LIN {X 0,Y 504.867,Z 563.28,A -85,B 0,C 180,E1 5576.571,E2 5576.571} C_VEL
LIN {X 0,Y 504.82,Z 563.28,A -85,B 0,C 180,E1 5581.711,E2 5581.711} C_VEL
LIN {X 0,Y 504.782,Z 563.28,A -85,B 0,C 180,E1 5586.866,E2 5586.866} C_VEL
LIN {X 0,Y 504.734,Z 563.28,A -85,B 0,C 180,E1 5592.078,E2 5592.078} C_VEL
LIN {X 0,Y 504.643,Z 563.28,A -85,B 0,C 180,E1 5597.397,E2 5597.397} C_VEL
LIN {X 0,Y 504.494,Z 563.28,A -85,B 0,C 180,E1 5602.88,E2 5602.88} C_VEL
LIN {X 0,Y 504.391,Z 563.28,A -85,B 0,C 180,E1 5608.597,E2 5608.597} C_VEL
LIN {X 0,Y 504.485,Z 563.28,A -85,B 0,C 180,E1 5614.631,E2 5614.631} C_VEL
LIN {X 0,Y 504.229,Z 563.28,A -85,B 0,C 180,E1 5621.174,E2 5621.174} C_VEL
LIN {X 0,Y 504.156,Z 563.28,A -85,B 0,C 180,E1 5621.894,E2 5621.894} C_VEL
LIN {X 0,Y 500.156,Z 563.28,A -85,B 0,C 180,E1 5623.841,E2 5623.841} C_VEL
LIN {X 0,Y 496.221,Z 563.28,A -85,B 0,C 180,E1 5625.82,E2 5625.82} C_VEL
LIN {X 0,Y 496.453,Z 563.28,A -85,B 0,C 180,E1 5632.208,E2 5632.208} C_VEL
LIN {X 0,Y 496.52,Z 563.28,A -85,B 0,C 180,E1 5633.043,E2 5633.043} C_VEL
LIN {X 0,Y 514.224,Z 600.382,A -85,B 0,C 180,E1 5635.156,E2 5635.156} C_VEL
LIN {X 0,Y 512.783,Z 642.692,A -85,B 0,C 180,E1 5636.234,E2 5636.234} C_VEL
LIN {X 0,Y 510.259,Z 681.705,A -85,B 0,C 180,E1 5637.958,E2 5637.958} C_VEL
LIN {X 0,Y 507.477,Z 717.491,A -85,B 0,C 180,E1 5640.249,E2 5640.249} C_VEL
LIN {X 0,Y 504.31,Z 752.435,A -85,B 0,C 180,E1 5643.33,E2 5643.33} C_VEL
LIN {X 0,Y 501.653,Z 781.389,A -85,B 0,C 180,E1 5646.722,E2 5646.722} C_VEL
LIN {X 0,Y 499.587,Z 807.919,A -85,B 0,C 180,E1 5650.823,E2 5650.823} C_VEL
LIN {X 0,Y 498.227,Z 828.231,A -85,B 0,C 180,E1 5655.074,E2 5655.074} C_VEL
LIN {X 0,Y 497.609,Z 843.281,A -85,B 0,C 180,E1 5659.516,E2 5659.516} C_VEL
LIN {X 0,Y 497.334,Z 852.705,A -85,B 0,C 180,E1 5663.903,E2 5663.903} C_VEL
LIN {X 0,Y 497.217,Z 857.111,A -85,B 0,C 180,E1 5668.26,E2 5668.26} C_VEL
LIN {X 0,Y 497.291,Z 857.112,A -85,B 0,C 180,E1 5671.738,E2 5671.738} C_VEL
LIN {X 0,Y 497.33,Z 852.707,A -85,B 0,C 180,E1 5676.095,E2 5676.095} C_VEL
LIN {X 0,Y 497.429,Z 843.286,A -85,B 0,C 180,E1 5680.486,E2 5680.486} C_VEL
LIN {X 0,Y 498.149,Z 828.634,A -85,B 0,C 180,E1 5684.83,E2 5684.83} C_VEL
LIN {X 0,Y 499.508,Z 807.928,A -85,B 0,C 180,E1 5689.179,E2 5689.179} C_VEL
LIN {X 0,Y 501.629,Z 781.403,A -85,B 0,C 180,E1 5693.277,E2 5693.277} C_VEL
LIN {X 0,Y 504.374,Z 751.392,A -85,B 0,C 180,E1 5696.775,E2 5696.775} C_VEL
LIN {X 0,Y 507.446,Z 717.513,A -85,B 0,C 180,E1 5699.751,E2 5699.751} C_VEL
LIN {X 0,Y 510.334,Z 680.807,A -85,B 0,C 180,E1 5702.09,E2 5702.09} C_VEL
LIN {X 0,Y 512.765,Z 641.796,A -85,B 0,C 180,E1 5703.799,E2 5703.799} C_VEL
LIN {X 0,Y 513.861,Z 600.092,A -85,B 0,C 180,E1 5704.878,E2 5704.878} C_VEL
LIN {X 0,Y 496.473,Z 563.28,A -85,B 0,C 180,E1 5707.017,E2 5707.017} C_VEL
LIN {X 0,Y 496.268,Z 563.28,A -85,B 0,C 180,E1 5713.136,E2 5713.136} C_VEL
LIN {X 0,Y 496.316,Z 563.28,A -85,B 0,C 180,E1 5719.472,E2 5719.472} C_VEL
LIN {X 0,Y 496.36,Z 563.28,A -85,B 0,C 180,E1 5725.168,E2 5725.168} C_VEL
LIN {X 0,Y 496.405,Z 563.28,A -85,B 0,C 180,E1 5731.83,E2 5731.83} C_VEL
LIN {X 0,Y 496.526,Z 563.28,A -85,B 0,C 180,E1 5736.731,E2 5736.731} C_VEL
LIN {X 0,Y 496.737,Z 563.28,A -85,B 0,C 180,E1 5742.317,E2 5742.317} C_VEL
LIN {X 0,Y 496.762,Z 563.28,A -85,B 0,C 180,E1 5749.501,E2 5749.501} C_VEL
LIN {X 0,Y 496.987,Z 563.28,A -85,B 0,C 180,E1 5754.776,E2 5754.776} C_VEL
LIN {X 0,Y 497.058,Z 563.28,A -85,B 0,C 180,E1 5760.002,E2 5760.002} C_VEL
LIN {X 0,Y 496.985,Z 563.28,A -85,B 0,C 180,E1 5765.228,E2 5765.228} C_VEL
LIN {X 0,Y 496.817,Z 563.28,A -85,B 0,C 180,E1 5770.502,E2 5770.502} C_VEL
LIN {X 0,Y 496.757,Z 563.28,A -85,B 0,C 180,E1 5775.868,E2 5775.868} C_VEL
LIN {X 0,Y 496.651,Z 563.28,A -85,B 0,C 180,E1 5781.385,E2 5781.385} C_VEL
LIN {X 0,Y 496.463,Z 563.28,A -85,B 0,C 180,E1 5787.126,E2 5787.126} C_VEL
LIN {X 0,Y 496.548,Z 563.28,A -85,B 0,C 180,E1 5793.164,E2 5793.164} C_VEL
LIN {X 0,Y 496.39,Z 563.28,A -85,B 0,C 180,E1 5799.674,E2 5799.674} C_VEL
LIN {X 0,Y 496.273,Z 563.28,A -85,B 0,C 180,E1 5805.626,E2 5805.626} C_VEL
LIN {X 0,Y 496.467,Z 563.28,A -85,B 0,C 180,E1 5812.212,E2 5812.212} C_VEL
LIN {X 0,Y 496.517,Z 563.28,A -85,B 0,C 180,E1 5818.32,E2 5818.32} C_VEL
LIN {X 0,Y 496.487,Z 563.28,A -85,B 0,C 180,E1 5824.818,E2 5824.818} C_VEL
LIN {X 0,Y 496.629,Z 563.28,A -85,B 0,C 180,E1 5830.475,E2 5830.475} C_VEL
LIN {X 0,Y 496.875,Z 563.28,A -85,B 0,C 180,E1 5836.375,E2 5836.375} C_VEL
LIN {X 0,Y 496.906,Z 563.28,A -85,B 0,C 180,E1 5841.267,E2 5841.267} C_VEL
LIN {X 0,Y 497.111,Z 563.28,A -85,B 0,C 180,E1 5846.52,E2 5846.52} C_VEL
LIN {X 0,Y 497.235,Z 563.28,A -85,B 0,C 180,E1 5851.74,E2 5851.74} C_VEL
LIN {X 0,Y 496.994,Z 563.28,A -85,B 0,C 180,E1 5856.977,E2 5856.977} C_VEL
LIN {X 0,Y 496.771,Z 563.28,A -85,B 0,C 180,E1 5863.576,E2 5863.576} C_VEL
LIN {X 0,Y 496.648,Z 563.28,A -85,B 0,C 180,E1 5869.624,E2 5869.624} C_VEL
LIN {X 0,Y 496.506,Z 563.28,A -85,B 0,C 180,E1 5875.183,E2 5875.183} C_VEL
LIN {X 0,Y 496.317,Z 563.28,A -85,B 0,C 180,E1 5881.643,E2 5881.643} C_VEL
LIN {X 0,Y 496.45,Z 563.28,A -85,B 0,C 180,E1 5887.785,E2 5887.785} C_VEL
LIN {X 0,Y 496.341,Z 563.28,A -85,B 0,C 180,E1 5894.369,E2 5894.369} C_VEL
LIN {X 0,Y 496.34,Z 563.28,A -85,B 0,C 180,E1 5900.322,E2 5900.322} C_VEL
LIN {X 0,Y 496.337,Z 563.28,A -85,B 0,C 180,E1 5906.82,E2 5906.82} C_VEL
LIN {X 0,Y 496.455,Z 563.28,A -85,B 0,C 180,E1 5912.873,E2 5912.873} C_VEL
LIN {X 0,Y 496.667,Z 563.28,A -85,B 0,C 180,E1 5918.616,E2 5918.616} C_VEL
LIN {X 0,Y 496.65,Z 563.28,A -85,B 0,C 180,E1 5924.128,E2 5924.128} C_VEL
LIN {X 0,Y 496.761,Z 563.28,A -85,B 0,C 180,E1 5929.497,E2 5929.497} C_VEL
LIN {X 0,Y 497.004,Z 563.28,A -85,B 0,C 180,E1 5934.772,E2 5934.772} C_VEL
LIN {X 0,Y 497.072,Z 563.28,A -85,B 0,C 180,E1 5939.998,E2 5939.998} C_VEL
LIN {X 0,Y 496.994,Z 563.28,A -85,B 0,C 180,E1 5945.224,E2 5945.224} C_VEL
LIN {X 0,Y 496.867,Z 563.28,A -85,B 0,C 180,E1 5950.497,E2 5950.497} C_VEL
LIN {X 0,Y 496.741,Z 563.28,A -85,B 0,C 180,E1 5955.865,E2 5955.865} C_VEL
LIN {X 0,Y 496.644,Z 563.28,A -85,B 0,C 180,E1 5961.381,E2 5961.381} C_VEL
LIN {X 0,Y 496.455,Z 563.28,A -85,B 0,C 180,E1 5967.123,E2 5967.123} C_VEL
LIN {X 0,Y 496.554,Z 563.28,A -85,B 0,C 180,E1 5973.16,E2 5973.16} C_VEL
LIN {X 0,Y 496.352,Z 563.28,A -85,B 0,C 180,E1 5979.673,E2 5979.673} C_VEL
LIN {X 0,Y 496.221,Z 563.28,A -85,B 0,C 180,E1 5985.82,E2 5985.82} C_VEL
LIN {X 0,Y 492.298,Z 563.28,A -85,B 0,C 180,E1 5987.795,E2 5987.795} C_VEL
LIN {X 0,Y 488.41,Z 563.28,A -85,B 0,C 180,E1 5989.801,E2 5989.801} C_VEL
LIN {X 0,Y 488.571,Z 563.784,A -85,B 0,C 180,E1 5992.379,E2 5992.379} C_VEL
LIN {X 0,Y 507.767,Z 604.447,A -85,B 0,C 180,E1 5994.736,E2 5994.736} C_VEL
LIN {X 0,Y 506.121,Z 643.782,A -85,B 0,C 180,E1 5995.777,E2 5995.777} C_VEL
LIN {X 0,Y 503.313,Z 683.897,A -85,B 0,C 180,E1 5997.593,E2 5997.593} C_VEL
LIN {X 0,Y 500.324,Z 718.929,A -85,B 0,C 180,E1 5999.905,E2 5999.905} C_VEL
LIN {X 0,Y 496.964,Z 753.499,A -85,B 0,C 180,E1 6003.018,E2 6003.018} C_VEL
LIN {X 0,Y 494.007,Z 783.215,A -85,B 0,C 180,E1 6006.602,E2 6006.602} C_VEL
LIN {X 0,Y 491.844,Z 807.92,A -85,B 0,C 180,E1 6010.509,E2 6010.509} C_VEL
LIN {X 0,Y 490.4,Z 828.252,A -85,B 0,C 180,E1 6014.837,E2 6014.837} C_VEL
LIN {X 0,Y 489.736,Z 843.28,A -85,B 0,C 180,E1 6019.345,E2 6019.345} C_VEL
LIN {X 0,Y 489.443,Z 852.701,A -85,B 0,C 180,E1 6023.804,E2 6023.804} C_VEL
LIN {X 0,Y 489.315,Z 857.112,A -85,B 0,C 180,E1 6028.232,E2 6028.232} C_VEL
LIN {X 0,Y 489.385,Z 857.113,A -85,B 0,C 180,E1 6031.766,E2 6031.766} C_VEL
LIN {X 0,Y 489.435,Z 852.703,A -85,B 0,C 180,E1 6036.194,E2 6036.194} C_VEL
LIN {X 0,Y 489.564,Z 843.284,A -85,B 0,C 180,E1 6040.657,E2 6040.657} C_VEL
LIN {X 0,Y 490.259,Z 830.078,A -85,B 0,C 180,E1 6044.71,E2 6044.71} C_VEL
LIN {X 0,Y 491.631,Z 810.331,A -85,B 0,C 180,E1 6049.033,E2 6049.033} C_VEL
LIN {X 0,Y 493.663,Z 786.566,A -85,B 0,C 180,E1 6052.937,E2 6052.937} C_VEL
LIN {X 0,Y 496.595,Z 756.593,A -85,B 0,C 180,E1 6056.655,E2 6056.655} C_VEL
LIN {X 0,Y 499.865,Z 723.287,A -85,B 0,C 180,E1 6059.749,E2 6059.749} C_VEL
LIN {X 0,Y 503.147,Z 687.121,A -85,B 0,C 180,E1 6062.227,E2 6062.227} C_VEL
LIN {X 0,Y 505.785,Z 649.282,A -85,B 0,C 180,E1 6064.01,E2 6064.01} C_VEL
LIN {X 0,Y 507.694,Z 611.444,A -85,B 0,C 180,E1 6065.125,E2 6065.125} C_VEL
LIN {X 0,Y 507.191,Z 602.422,A -85,B 0,C 180,E1 6065.351,E2 6065.351} C_VEL
LIN {X 0,Y 488.543,Z 563.28,A -85,B 0,C 180,E1 6067.702,E2 6067.702} C_VEL
LIN {X 0,Y 488.399,Z 563.28,A -85,B 0,C 180,E1 6074.717,E2 6074.717} C_VEL
LIN {X 0,Y 488.385,Z 563.28,A -85,B 0,C 180,E1 6080.573,E2 6080.573} C_VEL
LIN {X 0,Y 488.423,Z 563.28,A -85,B 0,C 180,E1 6086.529,E2 6086.529} C_VEL
LIN {X 0,Y 488.502,Z 563.28,A -85,B 0,C 180,E1 6092.399,E2 6092.399} C_VEL
LIN {X 0,Y 488.681,Z 563.28,A -85,B 0,C 180,E1 6098.253,E2 6098.253} C_VEL
LIN {X 0,Y 488.72,Z 563.28,A -85,B 0,C 180,E1 6103.868,E2 6103.868} C_VEL
LIN {X 0,Y 488.839,Z 563.28,A -85,B 0,C 180,E1 6109.328,E2 6109.328} C_VEL
LIN {X 0,Y 489.075,Z 563.28,A -85,B 0,C 180,E1 6114.691,E2 6114.691} C_VEL
LIN {X 0,Y 489.158,Z 563.28,A -85,B 0,C 180,E1 6120.002,E2 6120.002} C_VEL
LIN {X 0,Y 489.069,Z 563.28,A -85,B 0,C 180,E1 6125.313,E2 6125.313} C_VEL
LIN {X 0,Y 488.899,Z 563.28,A -85,B 0,C 180,E1 6130.674,E2 6130.674} C_VEL
LIN {X 0,Y 488.786,Z 563.28,A -85,B 0,C 180,E1 6136.856,E2 6136.856} C_VEL
LIN {X 0,Y 488.676,Z 563.28,A -85,B 0,C 180,E1 6142.124,E2 6142.124} C_VEL
LIN {X 0,Y 488.545,Z 563.28,A -85,B 0,C 180,E1 6147.603,E2 6147.603} C_VEL
LIN {X 0,Y 488.608,Z 563.28,A -85,B 0,C 180,E1 6153.775,E2 6153.775} C_VEL
LIN {X 0,Y 488.471,Z 563.28,A -85,B 0,C 180,E1 6159.439,E2 6159.439} C_VEL
LIN {X 0,Y 488.365,Z 563.28,A -85,B 0,C 180,E1 6165.292,E2 6165.292} C_VEL
LIN {X 0,Y 488.529,Z 563.28,A -85,B 0,C 180,E1 6171.847,E2 6171.847} C_VEL
LIN {X 0,Y 488.618,Z 563.28,A -85,B 0,C 180,E1 6178.332,E2 6178.332} C_VEL
LIN {X 0,Y 488.526,Z 563.28,A -85,B 0,C 180,E1 6184.378,E2 6184.378} C_VEL
LIN {X 0,Y 488.714,Z 563.28,A -85,B 0,C 180,E1 6190.145,E2 6190.145} C_VEL
LIN {X 0,Y 488.91,Z 563.28,A -85,B 0,C 180,E1 6195.706,E2 6195.706} C_VEL
LIN {X 0,Y 489.001,Z 563.28,A -85,B 0,C 180,E1 6201.125,E2 6201.125} C_VEL
LIN {X 0,Y 489.2,Z 563.28,A -85,B 0,C 180,E1 6206.464,E2 6206.464} C_VEL
LIN {X 0,Y 489.324,Z 563.28,A -85,B 0,C 180,E1 6211.768,E2 6211.768} C_VEL
LIN {X 0,Y 489.068,Z 563.28,A -85,B 0,C 180,E1 6217.09,E2 6217.09} C_VEL
LIN {X 0,Y 488.878,Z 563.28,A -85,B 0,C 180,E1 6222.479,E2 6222.479} C_VEL
LIN {X 0,Y 488.759,Z 563.28,A -85,B 0,C 180,E1 6227.984,E2 6227.984} C_VEL
LIN {X 0,Y 488.634,Z 563.28,A -85,B 0,C 180,E1 6233.671,E2 6233.671} C_VEL
LIN {X 0,Y 488.384,Z 563.28,A -85,B 0,C 180,E1 6240.099,E2 6240.099} C_VEL
LIN {X 0,Y 488.463,Z 563.28,A -85,B 0,C 180,E1 6245.943,E2 6245.943} C_VEL
LIN {X 0,Y 488.394,Z 563.28,A -85,B 0,C 180,E1 6252.136,E2 6252.136} C_VEL
LIN {X 0,Y 488.423,Z 563.28,A -85,B 0,C 180,E1 6257.86,E2 6257.86} C_VEL
LIN {X 0,Y 488.396,Z 563.28,A -85,B 0,C 180,E1 6264.051,E2 6264.051} C_VEL
LIN {X 0,Y 488.431,Z 563.28,A -85,B 0,C 180,E1 6270.373,E2 6270.373} C_VEL
LIN {X 0,Y 488.653,Z 563.28,A -85,B 0,C 180,E1 6276.329,E2 6276.329} C_VEL
LIN {X 0,Y 488.83,Z 563.28,A -85,B 0,C 180,E1 6282.018,E2 6282.018} C_VEL
LIN {X 0,Y 488.84,Z 563.28,A -85,B 0,C 180,E1 6289.325,E2 6289.325} C_VEL
LIN {X 0,Y 489.092,Z 563.28,A -85,B 0,C 180,E1 6294.687,E2 6294.687} C_VEL
LIN {X 0,Y 489.171,Z 563.28,A -85,B 0,C 180,E1 6299.998,E2 6299.998} C_VEL
LIN {X 0,Y 489.078,Z 563.28,A -85,B 0,C 180,E1 6305.309,E2 6305.309} C_VEL
LIN {X 0,Y 488.942,Z 563.28,A -85,B 0,C 180,E1 6310.669,E2 6310.669} C_VEL
LIN {X 0,Y 488.761,Z 563.28,A -85,B 0,C 180,E1 6316.841,E2 6316.841} C_VEL
LIN {X 0,Y 488.666,Z 563.28,A -85,B 0,C 180,E1 6322.116,E2 6322.116} C_VEL
LIN {X 0,Y 488.537,Z 563.28,A -85,B 0,C 180,E1 6327.599,E2 6327.599} C_VEL
LIN {X 0,Y 488.612,Z 563.28,A -85,B 0,C 180,E1 6333.77,E2 6333.77} C_VEL
LIN {X 0,Y 488.435,Z 563.28,A -85,B 0,C 180,E1 6339.432,E2 6339.432} C_VEL
LIN {X 0,Y 488.281,Z 563.28,A -85,B 0,C 180,E1 6345.814,E2 6345.814} C_VEL
LIN {X 0,Y 488.41,Z 563.28,A -85,B 0,C 180,E1 6349.801,E2 6349.801} C_VEL
LIN {X 0,Y 487.978,Z 566.18,A -85,B 0,C 180,E1 6350.996,E2 6350.996} C_VEL
LIN {X 0,Y 488.177,Z 576.133,A -85,B 0,C 180,E1 6352.344,E2 6352.344} C_VEL
LIN {X 0,Y 490.346,Z 583.192,A -85,B 0,C 180,E1 6352.886,E2 6352.886} C_VEL
LIN {X 0,Y 501.242,Z 607.303,A -85,B 0,C 180,E1 6354.273,E2 6354.273} C_VEL
LIN {X 0,Y 499.283,Z 646.915,A -85,B 0,C 180,E1 6355.391,E2 6355.391} C_VEL
LIN {X 0,Y 496.205,Z 687.92,A -85,B 0,C 180,E1 6357.329,E2 6357.329} C_VEL
LIN {X 0,Y 492.71,Z 724.764,A -85,B 0,C 180,E1 6359.904,E2 6359.904} C_VEL
LIN {X 0,Y 489.37,Z 756.878,A -85,B 0,C 180,E1 6362.954,E2 6362.954} C_VEL
LIN {X 0,Y 486.217,Z 786.547,A -85,B 0,C 180,E1 6366.689,E2 6366.689} C_VEL
LIN {X 0,Y 483.93,Z 811.51,A -85,B 0,C 180,E1 6370.887,E2 6370.887} C_VEL
LIN {X 0,Y 482.505,Z 830.074,A -85,B 0,C 180,E1 6375.047,E2 6375.047} C_VEL
LIN {X 0,Y 481.795,Z 844.724,A -85,B 0,C 180,E1 6379.743,E2 6379.743} C_VEL
LIN {X 0,Y 481.41,Z 854.003,A -85,B 0,C 180,E1 6384.603,E2 6384.603} C_VEL
LIN {X 0,Y 481.427,Z 857.113,A -85,B 0,C 180,E1 6388.203,E2 6388.203} C_VEL
LIN {X 0,Y 481.485,Z 857.114,A -85,B 0,C 180,E1 6391.795,E2 6391.795} C_VEL
LIN {X 0,Y 481.55,Z 852.699,A -85,B 0,C 180,E1 6396.296,E2 6396.296} C_VEL
LIN {X 0,Y 481.701,Z 843.283,A -85,B 0,C 180,E1 6400.833,E2 6400.833} C_VEL
LIN {X 0,Y 482.465,Z 830.081,A -85,B 0,C 180,E1 6404.953,E2 6404.953} C_VEL
LIN {X 0,Y 484.091,Z 809.135,A -85,B 0,C 180,E1 6409.578,E2 6409.578} C_VEL
LIN {X 0,Y 486.353,Z 784.891,A -85,B 0,C 180,E1 6413.544,E2 6413.544} C_VEL
LIN {X 0,Y 489.526,Z 755.489,A -85,B 0,C 180,E1 6417.203,E2 6417.203} C_VEL
LIN {X 0,Y 493.015,Z 722.001,A -85,B 0,C 180,E1 6420.317,E2 6420.317} C_VEL
LIN {X 0,Y 496.415,Z 685.825,A -85,B 0,C 180,E1 6422.783,E2 6422.783} C_VEL
LIN {X 0,Y 499.341,Z 645.989,A -85,B 0,C 180,E1 6424.646,E2 6424.646} C_VEL
LIN {X 0,Y 500.914,Z 605.537,A -85,B 0,C 180,E1 6425.791,E2 6425.791} C_VEL
LIN {X 0,Y 480.578,Z 563.28,A -85,B 0,C 180,E1 6428.392,E2 6428.392} C_VEL
LIN {X 0,Y 480.437,Z 563.28,A -85,B 0,C 180,E1 6433.75,E2 6433.75} C_VEL
LIN {X 0,Y 480.462,Z 563.28,A -85,B 0,C 180,E1 6438.917,E2 6438.917} C_VEL
LIN {X 0,Y 480.44,Z 563.28,A -85,B 0,C 180,E1 6444.748,E2 6444.748} C_VEL
LIN {X 0,Y 480.493,Z 563.28,A -85,B 0,C 180,E1 6449.838,E2 6449.838} C_VEL
LIN {X 0,Y 480.662,Z 563.28,A -85,B 0,C 180,E1 6455.915,E2 6455.915} C_VEL
LIN {X 0,Y 480.872,Z 563.28,A -85,B 0,C 180,E1 6461.714,E2 6461.714} C_VEL
LIN {X 0,Y 480.785,Z 563.28,A -85,B 0,C 180,E1 6467.31,E2 6467.31} C_VEL
LIN {X 0,Y 481.133,Z 563.28,A -85,B 0,C 180,E1 6472.795,E2 6472.795} C_VEL
LIN {X 0,Y 481.416,Z 563.28,A -85,B 0,C 180,E1 6478.206,E2 6478.206} C_VEL
LIN {X 0,Y 481.297,Z 563.28,A -85,B 0,C 180,E1 6483.597,E2 6483.597} C_VEL
LIN {X 0,Y 481.064,Z 563.28,A -85,B 0,C 180,E1 6489.025,E2 6489.025} C_VEL
LIN {X 0,Y 480.976,Z 563.28,A -85,B 0,C 180,E1 6494.538,E2 6494.538} C_VEL
LIN {X 0,Y 480.827,Z 563.28,A -85,B 0,C 180,E1 6500.197,E2 6500.197} C_VEL
LIN {X 0,Y 480.651,Z 563.28,A -85,B 0,C 180,E1 6506.076,E2 6506.076} C_VEL
LIN {X 0,Y 480.66,Z 563.28,A -85,B 0,C 180,E1 6512.258,E2 6512.258} C_VEL
LIN {X 0,Y 480.585,Z 563.28,A -85,B 0,C 180,E1 6518.904,E2 6518.904} C_VEL
LIN {X 0,Y 480.406,Z 563.28,A -85,B 0,C 180,E1 6523.744,E2 6523.744} C_VEL
LIN {X 0,Y 480.469,Z 563.28,A -85,B 0,C 180,E1 6528.92,E2 6528.92} C_VEL
LIN {X 0,Y 480.628,Z 563.28,A -85,B 0,C 180,E1 6534.719,E2 6534.719} C_VEL
LIN {X 0,Y 480.653,Z 563.28,A -85,B 0,C 180,E1 6539.847,E2 6539.847} C_VEL
LIN {X 0,Y 480.604,Z 563.28,A -85,B 0,C 180,E1 6545.911,E2 6545.911} C_VEL
LIN {X 0,Y 480.82,Z 563.28,A -85,B 0,C 180,E1 6551.71,E2 6551.71} C_VEL
LIN {X 0,Y 481.01,Z 563.28,A -85,B 0,C 180,E1 6557.315,E2 6557.315} C_VEL
LIN {X 0,Y 481.09,Z 563.28,A -85,B 0,C 180,E1 6562.793,E2 6562.793} C_VEL
LIN {X 0,Y 481.194,Z 563.28,A -85,B 0,C 180,E1 6568.204,E2 6568.204} C_VEL
LIN {X 0,Y 481.212,Z 563.28,A -85,B 0,C 180,E1 6573.597,E2 6573.597} C_VEL
LIN {X 0,Y 481.043,Z 563.28,A -85,B 0,C 180,E1 6579.025,E2 6579.025} C_VEL
LIN {X 0,Y 480.919,Z 563.28,A -85,B 0,C 180,E1 6584.539,E2 6584.539} C_VEL
LIN {X 0,Y 480.787,Z 563.28,A -85,B 0,C 180,E1 6590.198,E2 6590.198} C_VEL
LIN {X 0,Y 480.615,Z 563.28,A -85,B 0,C 180,E1 6596.077,E2 6596.077} C_VEL
LIN {X 0,Y 480.505,Z 563.28,A -85,B 0,C 180,E1 6602.269,E2 6602.269} C_VEL
LIN {X 0,Y 480.583,Z 563.28,A -85,B 0,C 180,E1 6608.903,E2 6608.903} C_VEL
LIN {X 0,Y 480.47,Z 563.28,A -85,B 0,C 180,E1 6613.749,E2 6613.749} C_VEL
LIN {X 0,Y 480.48,Z 563.28,A -85,B 0,C 180,E1 6618.918,E2 6618.918} C_VEL
LIN {X 0,Y 480.443,Z 563.28,A -85,B 0,C 180,E1 6624.75,E2 6624.75} C_VEL
LIN {X 0,Y 480.501,Z 563.28,A -85,B 0,C 180,E1 6629.834,E2 6629.834} C_VEL
LIN {X 0,Y 480.686,Z 563.28,A -85,B 0,C 180,E1 6635.912,E2 6635.912} C_VEL
LIN {X 0,Y 480.889,Z 563.28,A -85,B 0,C 180,E1 6641.71,E2 6641.71} C_VEL
LIN {X 0,Y 480.775,Z 563.28,A -85,B 0,C 180,E1 6647.306,E2 6647.306} C_VEL
LIN {X 0,Y 481.112,Z 563.28,A -85,B 0,C 180,E1 6653.004,E2 6653.004} C_VEL
LIN {X 0,Y 481.434,Z 563.28,A -85,B 0,C 180,E1 6658.202,E2 6658.202} C_VEL
LIN {X 0,Y 481.264,Z 563.28,A -85,B 0,C 180,E1 6663.593,E2 6663.593} C_VEL
LIN {X 0,Y 481.073,Z 563.28,A -85,B 0,C 180,E1 6669.021,E2 6669.021} C_VEL
LIN {X 0,Y 480.971,Z 563.28,A -85,B 0,C 180,E1 6674.534,E2 6674.534} C_VEL
LIN {X 0,Y 480.819,Z 563.28,A -85,B 0,C 180,E1 6680.193,E2 6680.193} C_VEL
LIN {X 0,Y 480.639,Z 563.28,A -85,B 0,C 180,E1 6686.072,E2 6686.072} C_VEL
LIN {X 0,Y 480.658,Z 563.28,A -85,B 0,C 180,E1 6692.254,E2 6692.254} C_VEL
LIN {X 0,Y 480.607,Z 563.28,A -85,B 0,C 180,E1 6698.283,E2 6698.283} C_VEL
LIN {X 0,Y 480.373,Z 563.28,A -85,B 0,C 180,E1 6703.737,E2 6703.737} C_VEL
LIN {X 0,Y 480.416,Z 563.28,A -85,B 0,C 180,E1 6709.804,E2 6709.804} C_VEL
LIN {X 0,Y 480.623,Z 564,A -85,B 0,C 180,E1 6711.655,E2 6711.655} C_VEL
LIN {X 0,Y 490.346,Z 583.192,A -85,B 0,C 180,E1 6712.886,E2 6712.886} C_VEL
LIN {X 0,Y 493.821,Z 595.133,A -85,B 0,C 180,E1 6713.4,E2 6713.4} C_VEL
LIN {X 0,Y 494.395,Z 616.987,A -85,B 0,C 180,E1 6713.952,E2 6713.952} C_VEL
LIN {X 0,Y 491.949,Z 657.63,A -85,B 0,C 180,E1 6715.296,E2 6715.296} C_VEL
LIN {X 0,Y 488.506,Z 697.035,A -85,B 0,C 180,E1 6717.407,E2 6717.407} C_VEL
LIN {X 0,Y 484.975,Z 731.703,A -85,B 0,C 180,E1 6720.03,E2 6720.03} C_VEL
LIN {X 0,Y 481.133,Z 765.214,A -85,B 0,C 180,E1 6723.468,E2 6723.468} C_VEL
LIN {X 0,Y 478.108,Z 792.986,A -85,B 0,C 180,E1 6727.3,E2 6727.3} C_VEL
LIN {X 0,Y 475.843,Z 816.208,A -85,B 0,C 180,E1 6731.51,E2 6731.51} C_VEL
LIN {X 0,Y 474.304,Z 835.931,A -85,B 0,C 180,E1 6736.472,E2 6736.472} C_VEL
LIN {X 0,Y 473.778,Z 847.752,A -85,B 0,C 180,E1 6740.865,E2 6740.865} C_VEL
LIN {X 0,Y 473.521,Z 854.003,A -85,B 0,C 180,E1 6744.513,E2 6744.513} C_VEL
LIN {X 0,Y 473.524,Z 857.113,A -85,B 0,C 180,E1 6748.173,E2 6748.173} C_VEL
LIN {X 0,Y 473.579,Z 857.114,A -85,B 0,C 180,E1 6751.825,E2 6751.825} C_VEL
LIN {X 0,Y 473.641,Z 852.696,A -85,B 0,C 180,E1 6756.401,E2 6756.401} C_VEL
LIN {X 0,Y 473.865,Z 843.282,A -85,B 0,C 180,E1 6761.014,E2 6761.014} C_VEL
LIN {X 0,Y 474.677,Z 830.084,A -85,B 0,C 180,E1 6765.204,E2 6765.204} C_VEL
LIN {X 0,Y 476.439,Z 809.132,A -85,B 0,C 180,E1 6769.905,E2 6769.905} C_VEL
LIN {X 0,Y 478.97,Z 784.467,A -85,B 0,C 180,E1 6773.991,E2 6773.991} C_VEL
LIN {X 0,Y 482.347,Z 755.059,A -85,B 0,C 180,E1 6777.694,E2 6777.694} C_VEL
LIN {X 0,Y 486.177,Z 720.586,A -85,B 0,C 180,E1 6780.895,E2 6780.895} C_VEL
LIN {X 0,Y 489.749,Z 684.504,A -85,B 0,C 180,E1 6783.352,E2 6783.352} C_VEL
LIN {X 0,Y 492.928,Z 643.347,A -85,B 0,C 180,E1 6785.27,E2 6785.27} C_VEL
LIN {X 0,Y 494.202,Z 607.589,A -85,B 0,C 180,E1 6786.305,E2 6786.305} C_VEL
LIN {X 0,Y 472.752,Z 564.557,A -85,B 0,C 180,E1 6789.087,E2 6789.087} C_VEL
LIN {X 0,Y 472.592,Z 563.28,A -85,B 0,C 180,E1 6789.255,E2 6789.255} C_VEL
LIN {X 0,Y 472.456,Z 563.28,A -85,B 0,C 180,E1 6795.362,E2 6795.362} C_VEL
LIN {X 0,Y 472.499,Z 563.28,A -85,B 0,C 180,E1 6800.306,E2 6800.306} C_VEL
LIN {X 0,Y 472.498,Z 563.28,A -85,B 0,C 180,E1 6806.134,E2 6806.134} C_VEL
LIN {X 0,Y 472.615,Z 563.28,A -85,B 0,C 180,E1 6811.387,E2 6811.387} C_VEL
LIN {X 0,Y 472.85,Z 563.28,A -85,B 0,C 180,E1 6817.738,E2 6817.738} C_VEL
LIN {X 0,Y 472.904,Z 563.28,A -85,B 0,C 180,E1 6823.313,E2 6823.313} C_VEL
LIN {X 0,Y 472.97,Z 563.28,A -85,B 0,C 180,E1 6828.966,E2 6828.966} C_VEL
LIN {X 0,Y 473.25,Z 563.28,A -85,B 0,C 180,E1 6834.513,E2 6834.513} C_VEL
LIN {X 0,Y 473.363,Z 563.28,A -85,B 0,C 180,E1 6840.002,E2 6840.002} C_VEL
LIN {X 0,Y 473.237,Z 563.28,A -85,B 0,C 180,E1 6845.491,E2 6845.491} C_VEL
LIN {X 0,Y 473.06,Z 563.28,A -85,B 0,C 180,E1 6851.036,E2 6851.036} C_VEL
LIN {X 0,Y 472.956,Z 563.28,A -85,B 0,C 180,E1 6856.831,E2 6856.831} C_VEL
LIN {X 0,Y 472.824,Z 563.28,A -85,B 0,C 180,E1 6862.52,E2 6862.52} C_VEL
LIN {X 0,Y 472.687,Z 563.28,A -85,B 0,C 180,E1 6868.613,E2 6868.613} C_VEL
LIN {X 0,Y 472.727,Z 563.28,A -85,B 0,C 180,E1 6875.072,E2 6875.072} C_VEL
LIN {X 0,Y 472.543,Z 563.28,A -85,B 0,C 180,E1 6879.969,E2 6879.969} C_VEL
LIN {X 0,Y 472.424,Z 563.28,A -85,B 0,C 180,E1 6885.356,E2 6885.356} C_VEL
LIN {X 0,Y 472.563,Z 563.28,A -85,B 0,C 180,E1 6890.31,E2 6890.31} C_VEL
LIN {X 0,Y 472.693,Z 563.28,A -85,B 0,C 180,E1 6896.102,E2 6896.102} C_VEL
LIN {X 0,Y 472.694,Z 563.28,A -85,B 0,C 180,E1 6901.39,E2 6901.39} C_VEL
LIN {X 0,Y 472.769,Z 563.28,A -85,B 0,C 180,E1 6907.767,E2 6907.767} C_VEL
LIN {X 0,Y 472.953,Z 563.28,A -85,B 0,C 180,E1 6913.313,E2 6913.313} C_VEL
LIN {X 0,Y 473.118,Z 563.28,A -85,B 0,C 180,E1 6918.968,E2 6918.968} C_VEL
LIN {X 0,Y 473.254,Z 563.28,A -85,B 0,C 180,E1 6924.512,E2 6924.512} C_VEL
LIN {X 0,Y 473.373,Z 563.28,A -85,B 0,C 180,E1 6930.001,E2 6930.001} C_VEL
LIN {X 0,Y 473.297,Z 563.28,A -85,B 0,C 180,E1 6935.49,E2 6935.49} C_VEL
LIN {X 0,Y 473.051,Z 563.28,A -85,B 0,C 180,E1 6941.035,E2 6941.035} C_VEL
LIN {X 0,Y 472.911,Z 563.28,A -85,B 0,C 180,E1 6946.807,E2 6946.807} C_VEL
LIN {X 0,Y 472.814,Z 563.28,A -85,B 0,C 180,E1 6952.52,E2 6952.52} C_VEL
LIN {X 0,Y 472.573,Z 563.28,A -85,B 0,C 180,E1 6958.62,E2 6958.62} C_VEL
LIN {X 0,Y 472.624,Z 563.28,A -85,B 0,C 180,E1 6965.08,E2 6965.08} C_VEL
LIN {X 0,Y 472.545,Z 563.28,A -85,B 0,C 180,E1 6969.966,E2 6969.966} C_VEL
LIN {X 0,Y 472.489,Z 563.28,A -85,B 0,C 180,E1 6975.36,E2 6975.36} C_VEL
LIN {X 0,Y 472.522,Z 563.28,A -85,B 0,C 180,E1 6980.303,E2 6980.303} C_VEL
LIN {X 0,Y 472.516,Z 563.28,A -85,B 0,C 180,E1 6986.134,E2 6986.134} C_VEL
LIN {X 0,Y 472.629,Z 563.28,A -85,B 0,C 180,E1 6991.383,E2 6991.383} C_VEL
LIN {X 0,Y 472.869,Z 563.28,A -85,B 0,C 180,E1 6997.737,E2 6997.737} C_VEL
LIN {X 0,Y 472.92,Z 563.28,A -85,B 0,C 180,E1 7003.309,E2 7003.309} C_VEL
LIN {X 0,Y 472.968,Z 563.28,A -85,B 0,C 180,E1 7008.962,E2 7008.962} C_VEL
LIN {X 0,Y 473.265,Z 563.28,A -85,B 0,C 180,E1 7014.509,E2 7014.509} C_VEL
LIN {X 0,Y 473.375,Z 563.28,A -85,B 0,C 180,E1 7019.998,E2 7019.998} C_VEL
LIN {X 0,Y 473.245,Z 563.28,A -85,B 0,C 180,E1 7025.487,E2 7025.487} C_VEL
LIN {X 0,Y 473.117,Z 563.28,A -85,B 0,C 180,E1 7031.031,E2 7031.031} C_VEL
LIN {X 0,Y 472.935,Z 563.28,A -85,B 0,C 180,E1 7036.817,E2 7036.817} C_VEL
LIN {X 0,Y 472.815,Z 563.28,A -85,B 0,C 180,E1 7042.516,E2 7042.516} C_VEL
LIN {X 0,Y 472.681,Z 563.28,A -85,B 0,C 180,E1 7048.609,E2 7048.609} C_VEL
LIN {X 0,Y 472.725,Z 563.28,A -85,B 0,C 180,E1 7055.068,E2 7055.068} C_VEL
LIN {X 0,Y 472.515,Z 563.28,A -85,B 0,C 180,E1 7059.962,E2 7059.962} C_VEL
LIN {X 0,Y 472.393,Z 563.28,A -85,B 0,C 180,E1 7065.349,E2 7065.349} C_VEL
LIN {X 0,Y 472.65,Z 563.28,A -85,B 0,C 180,E1 7070.865,E2 7070.865} C_VEL
LIN {X 0,Y 477.303,Z 573.451,A -85,B 0,C 180,E1 7071.519,E2 7071.519} C_VEL
LIN {X 0,Y 494.783,Z 608.873,A -85,B 0,C 180,E1 7073.772,E2 7073.772} C_VEL
LIN {X 0,Y 494.395,Z 616.987,A -85,B 0,C 180,E1 7073.952,E2 7073.952} C_VEL
LIN {X 0,Y 490.198,Z 633.953,A -85,B 0,C 180,E1 7074.153,E2 7074.153} C_VEL
LIN {X 0,Y 486.085,Z 648.568,A -85,B 0,C 180,E1 7074.409,E2 7074.409} C_VEL
LIN {X 0,Y 485.874,Z 650.65,A -85,B 0,C 180,E1 7074.488,E2 7074.488} C_VEL
LIN {X 0,Y 482.703,Z 687.757,A -85,B 0,C 180,E1 7076.318,E2 7076.318} C_VEL
LIN {X 0,Y 478.72,Z 724.66,A -85,B 0,C 180,E1 7078.961,E2 7078.961} C_VEL
LIN {X 0,Y 475.004,Z 756.172,A -85,B 0,C 180,E1 7081.999,E2 7081.999} C_VEL
LIN {X 0,Y 471.409,Z 785.703,A -85,B 0,C 180,E1 7085.786,E2 7085.786} C_VEL
LIN {X 0,Y 468.622,Z 810.311,A -85,B 0,C 180,E1 7089.992,E2 7089.992} C_VEL
LIN {X 0,Y 466.898,Z 830.081,A -85,B 0,C 180,E1 7094.535,E2 7094.535} C_VEL
LIN {X 0,Y 466.069,Z 844.423,A -85,B 0,C 180,E1 7099.27,E2 7099.27} C_VEL
LIN {X 0,Y 465.745,Z 852.689,A -85,B 0,C 180,E1 7103.488,E2 7103.488} C_VEL
LIN {X 0,Y 465.624,Z 857.113,A -85,B 0,C 180,E1 7108.142,E2 7108.142} C_VEL
LIN {X 0,Y 465.671,Z 857.113,A -85,B 0,C 180,E1 7111.856,E2 7111.856} C_VEL
LIN {X 0,Y 465.734,Z 852.692,A -85,B 0,C 180,E1 7116.511,E2 7116.511} C_VEL
LIN {X 0,Y 466.004,Z 843.281,A -85,B 0,C 180,E1 7121.202,E2 7121.202} C_VEL
LIN {X 0,Y 467.081,Z 828.244,A -85,B 0,C 180,E1 7125.938,E2 7125.938} C_VEL
LIN {X 0,Y 468.919,Z 807.932,A -85,B 0,C 180,E1 7130.484,E2 7130.484} C_VEL
LIN {X 0,Y 471.927,Z 781.539,A -85,B 0,C 180,E1 7134.813,E2 7134.813} C_VEL
LIN {X 0,Y 475.426,Z 752.23,A -85,B 0,C 180,E1 7138.43,E2 7138.43} C_VEL
LIN {X 0,Y 479.61,Z 716.853,A -85,B 0,C 180,E1 7141.682,E2 7141.682} C_VEL
LIN {X 0,Y 483.505,Z 678.903,A -85,B 0,C 180,E1 7144.178,E2 7144.178} C_VEL
LIN {X 0,Y 486.547,Z 640.865,A -85,B 0,C 180,E1 7145.891,E2 7145.891} C_VEL
LIN {X 0,Y 487.936,Z 610.645,A -85,B 0,C 180,E1 7146.775,E2 7146.775} C_VEL
LIN {X 0,Y 466.467,Z 568.331,A -85,B 0,C 180,E1 7149.638,E2 7149.638} C_VEL
LIN {X 0,Y 464.617,Z 563.28,A -85,B 0,C 180,E1 7149.926,E2 7149.926} C_VEL
LIN {X 0,Y 464.531,Z 563.28,A -85,B 0,C 180,E1 7155.614,E2 7155.614} C_VEL
LIN {X 0,Y 464.566,Z 563.28,A -85,B 0,C 180,E1 7161.894,E2 7161.894} C_VEL
LIN {X 0,Y 464.549,Z 563.28,A -85,B 0,C 180,E1 7167.624,E2 7167.624} C_VEL
LIN {X 0,Y 464.735,Z 563.28,A -85,B 0,C 180,E1 7172.964,E2 7172.964} C_VEL
LIN {X 0,Y 464.959,Z 563.28,A -85,B 0,C 180,E1 7179.086,E2 7179.086} C_VEL
LIN {X 0,Y 464.893,Z 563.28,A -85,B 0,C 180,E1 7184.952,E2 7184.952} C_VEL
LIN {X 0,Y 465.133,Z 563.28,A -85,B 0,C 180,E1 7190.667,E2 7190.667} C_VEL
LIN {X 0,Y 465.39,Z 563.28,A -85,B 0,C 180,E1 7196.284,E2 7196.284} C_VEL
LIN {X 0,Y 465.431,Z 563.28,A -85,B 0,C 180,E1 7201.86,E2 7201.86} C_VEL
LIN {X 0,Y 465.259,Z 563.28,A -85,B 0,C 180,E1 7207.456,E2 7207.456} C_VEL
LIN {X 0,Y 465.16,Z 563.28,A -85,B 0,C 180,E1 7213.294,E2 7213.294} C_VEL
LIN {X 0,Y 464.954,Z 563.28,A -85,B 0,C 180,E1 7219.749,E2 7219.749} C_VEL
LIN {X 0,Y 464.814,Z 563.28,A -85,B 0,C 180,E1 7224.965,E2 7224.965} C_VEL
LIN {X 0,Y 464.716,Z 563.28,A -85,B 0,C 180,E1 7231.304,E2 7231.304} C_VEL
LIN {X 0,Y 464.777,Z 563.28,A -85,B 0,C 180,E1 7235.763,E2 7235.763} C_VEL
LIN {X 0,Y 464.541,Z 563.28,A -85,B 0,C 180,E1 7241.659,E2 7241.659} C_VEL
LIN {X 0,Y 464.54,Z 563.28,A -85,B 0,C 180,E1 7248.344,E2 7248.344} C_VEL
LIN {X 0,Y 464.773,Z 563.28,A -85,B 0,C 180,E1 7254.264,E2 7254.264} C_VEL
LIN {X 0,Y 464.765,Z 563.28,A -85,B 0,C 180,E1 7260.856,E2 7260.856} C_VEL
LIN {X 0,Y 464.799,Z 563.28,A -85,B 0,C 180,E1 7267.072,E2 7267.072} C_VEL
LIN {X 0,Y 465.034,Z 563.28,A -85,B 0,C 180,E1 7273.021,E2 7273.021} C_VEL
LIN {X 0,Y 465.195,Z 563.28,A -85,B 0,C 180,E1 7278.778,E2 7278.778} C_VEL
LIN {X 0,Y 465.361,Z 563.28,A -85,B 0,C 180,E1 7284.418,E2 7284.418} C_VEL
LIN {X 0,Y 465.503,Z 563.28,A -85,B 0,C 180,E1 7290.001,E2 7290.001} C_VEL
LIN {X 0,Y 465.403,Z 563.28,A -85,B 0,C 180,E1 7295.583,E2 7295.583} C_VEL
LIN {X 0,Y 465.129,Z 563.28,A -85,B 0,C 180,E1 7301.226,E2 7301.226} C_VEL
LIN {X 0,Y 465.01,Z 563.28,A -85,B 0,C 180,E1 7306.982,E2 7306.982} C_VEL
LIN {X 0,Y 464.855,Z 563.28,A -85,B 0,C 180,E1 7312.927,E2 7312.927} C_VEL
LIN {X 0,Y 464.633,Z 563.28,A -85,B 0,C 180,E1 7319.155,E2 7319.155} C_VEL
LIN {X 0,Y 464.708,Z 563.28,A -85,B 0,C 180,E1 7325.769,E2 7325.769} C_VEL
LIN {X 0,Y 464.56,Z 563.28,A -85,B 0,C 180,E1 7331.658,E2 7331.658} C_VEL
LIN {X 0,Y 464.557,Z 563.28,A -85,B 0,C 180,E1 7338.341,E2 7338.341} C_VEL
LIN {X 0,Y 464.619,Z 563.28,A -85,B 0,C 180,E1 7344.289,E2 7344.289} C_VEL
LIN {X 0,Y 464.731,Z 563.28,A -85,B 0,C 180,E1 7351.249,E2 7351.249} C_VEL
LIN {X 0,Y 464.875,Z 563.28,A -85,B 0,C 180,E1 7357.073,E2 7357.073} C_VEL
LIN {X 0,Y 465.017,Z 563.28,A -85,B 0,C 180,E1 7363.017,E2 7363.017} C_VEL
LIN {X 0,Y 465.034,Z 563.28,A -85,B 0,C 180,E1 7368.771,E2 7368.771} C_VEL
LIN {X 0,Y 465.373,Z 563.28,A -85,B 0,C 180,E1 7374.416,E2 7374.416} C_VEL
LIN {X 0,Y 465.504,Z 563.28,A -85,B 0,C 180,E1 7379.998,E2 7379.998} C_VEL
LIN {X 0,Y 465.352,Z 563.28,A -85,B 0,C 180,E1 7385.581,E2 7385.581} C_VEL
LIN {X 0,Y 465.194,Z 563.28,A -85,B 0,C 180,E1 7391.221,E2 7391.221} C_VEL
LIN {X 0,Y 465.032,Z 563.28,A -85,B 0,C 180,E1 7396.978,E2 7396.978} C_VEL
LIN {X 0,Y 464.857,Z 563.28,A -85,B 0,C 180,E1 7402.923,E2 7402.923} C_VEL
LIN {X 0,Y 464.748,Z 563.28,A -85,B 0,C 180,E1 7409.144,E2 7409.144} C_VEL
LIN {X 0,Y 464.768,Z 563.28,A -85,B 0,C 180,E1 7415.759,E2 7415.759} C_VEL
LIN {X 0,Y 464.511,Z 563.28,A -85,B 0,C 180,E1 7421.652,E2 7421.652} C_VEL
LIN {X 0,Y 464.518,Z 563.28,A -85,B 0,C 180,E1 7428.342,E2 7428.342} C_VEL
LIN {X 0,Y 464.66,Z 563.28,A -85,B 0,C 180,E1 7430.067,E2 7430.067} C_VEL
LIN {X 0,Y 468.699,Z 572.337,A -85,B 0,C 180,E1 7430.663,E2 7430.663} C_VEL
LIN {X 0,Y 488.239,Z 610.762,A -85,B 0,C 180,E1 7433.254,E2 7433.254} C_VEL
LIN {X 0,Y 485.874,Z 650.65,A -85,B 0,C 180,E1 7434.488,E2 7434.488} C_VEL
LIN {X 0,Y 481.306,Z 667.263,A -85,B 0,C 180,E1 7434.96,E2 7434.96} C_VEL
LIN {X 0,Y 476.49,Z 683.237,A -85,B 0,C 180,E1 7435.543,E2 7435.543} C_VEL
LIN {X 0,Y 472.537,Z 718.445,A -85,B 0,C 180,E1 7437.958,E2 7437.958} C_VEL
LIN {X 0,Y 468.049,Z 754.278,A -85,B 0,C 180,E1 7441.341,E2 7441.341} C_VEL
LIN {X 0,Y 463.944,Z 785.89,A -85,B 0,C 180,E1 7445.413,E2 7445.413} C_VEL
LIN {X 0,Y 461.112,Z 809.116,A -85,B 0,C 180,E1 7449.402,E2 7449.402} C_VEL
LIN {X 0,Y 459.093,Z 830.082,A -85,B 0,C 180,E1 7454.265,E2 7454.265} C_VEL
LIN {X 0,Y 458.196,Z 844.422,A -85,B 0,C 180,E1 7459.083,E2 7459.083} C_VEL
LIN {X 0,Y 457.854,Z 852.685,A -85,B 0,C 180,E1 7463.375,E2 7463.375} C_VEL
LIN {X 0,Y 457.721,Z 857.112,A -85,B 0,C 180,E1 7468.11,E2 7468.11} C_VEL
LIN {X 0,Y 457.766,Z 857.113,A -85,B 0,C 180,E1 7471.888,E2 7471.888} C_VEL
LIN {X 0,Y 457.843,Z 852.688,A -85,B 0,C 180,E1 7476.623,E2 7476.623} C_VEL
LIN {X 0,Y 458.175,Z 843.279,A -85,B 0,C 180,E1 7481.396,E2 7481.396} C_VEL
LIN {X 0,Y 459.332,Z 828.239,A -85,B 0,C 180,E1 7486.214,E2 7486.214} C_VEL
LIN {X 0,Y 461.307,Z 807.933,A -85,B 0,C 180,E1 7490.838,E2 7490.838} C_VEL
LIN {X 0,Y 464.328,Z 783.087,A -85,B 0,C 180,E1 7494.991,E2 7494.991} C_VEL
LIN {X 0,Y 468.13,Z 753.141,A -85,B 0,C 180,E1 7498.783,E2 7498.783} C_VEL
LIN {X 0,Y 472.598,Z 717.611,A -85,B 0,C 180,E1 7502.114,E2 7502.114} C_VEL
LIN {X 0,Y 476.69,Z 680.564,A -85,B 0,C 180,E1 7504.613,E2 7504.613} C_VEL
LIN {X 0,Y 480.085,Z 641.296,A -85,B 0,C 180,E1 7506.424,E2 7506.424} C_VEL
LIN {X 0,Y 481.417,Z 613.029,A -85,B 0,C 180,E1 7507.286,E2 7507.286} C_VEL
LIN {X 0,Y 461.131,Z 573.058,A -85,B 0,C 180,E1 7510.091,E2 7510.091} C_VEL
LIN {X 0,Y 456.755,Z 564.588,A -85,B 0,C 180,E1 7510.723,E2 7510.723} C_VEL
LIN {X 0,Y 456.636,Z 563.28,A -85,B 0,C 180,E1 7510.863,E2 7510.863} C_VEL
LIN {X 0,Y 456.656,Z 563.28,A -85,B 0,C 180,E1 7516.633,E2 7516.633} C_VEL
LIN {X 0,Y 456.626,Z 563.28,A -85,B 0,C 180,E1 7523.502,E2 7523.502} C_VEL
LIN {X 0,Y 456.672,Z 563.28,A -85,B 0,C 180,E1 7530.29,E2 7530.29} C_VEL
LIN {X 0,Y 456.907,Z 563.28,A -85,B 0,C 180,E1 7536.654,E2 7536.654} C_VEL
LIN {X 0,Y 457.097,Z 563.28,A -85,B 0,C 180,E1 7543.208,E2 7543.208} C_VEL
LIN {X 0,Y 457.123,Z 563.28,A -85,B 0,C 180,E1 7548.578,E2 7548.578} C_VEL
LIN {X 0,Y 457.442,Z 563.28,A -85,B 0,C 180,E1 7554.323,E2 7554.323} C_VEL
LIN {X 0,Y 457.592,Z 563.28,A -85,B 0,C 180,E1 7560.002,E2 7560.002} C_VEL
LIN {X 0,Y 457.426,Z 563.28,A -85,B 0,C 180,E1 7565.682,E2 7565.682} C_VEL
LIN {X 0,Y 457.232,Z 563.28,A -85,B 0,C 180,E1 7571.423,E2 7571.423} C_VEL
LIN {X 0,Y 457.109,Z 563.28,A -85,B 0,C 180,E1 7577.286,E2 7577.286} C_VEL
LIN {X 0,Y 456.926,Z 563.28,A -85,B 0,C 180,E1 7583.349,E2 7583.349} C_VEL
LIN {X 0,Y 456.781,Z 563.28,A -85,B 0,C 180,E1 7589.707,E2 7589.707} C_VEL
LIN {X 0,Y 456.76,Z 563.28,A -85,B 0,C 180,E1 7596.491,E2 7596.491} C_VEL
LIN {X 0,Y 456.609,Z 563.28,A -85,B 0,C 180,E1 7603.361,E2 7603.361} C_VEL
LIN {X 0,Y 456.675,Z 563.28,A -85,B 0,C 180,E1 7609.466,E2 7609.466} C_VEL
LIN {X 0,Y 456.803,Z 563.28,A -85,B 0,C 180,E1 7615.836,E2 7615.836} C_VEL
LIN {X 0,Y 456.831,Z 563.28,A -85,B 0,C 180,E1 7622.456,E2 7622.456} C_VEL
LIN {X 0,Y 456.928,Z 563.28,A -85,B 0,C 180,E1 7628.699,E2 7628.699} C_VEL
LIN {X 0,Y 457.156,Z 563.28,A -85,B 0,C 180,E1 7634.689,E2 7634.689} C_VEL
LIN {X 0,Y 457.356,Z 563.28,A -85,B 0,C 180,E1 7640.505,E2 7640.505} C_VEL
LIN {X 0,Y 457.579,Z 563.28,A -85,B 0,C 180,E1 7646.219,E2 7646.219} C_VEL
LIN {X 0,Y 457.71,Z 563.28,A -85,B 0,C 180,E1 7651.89,E2 7651.89} C_VEL
LIN {X 0,Y 457.337,Z 563.28,A -85,B 0,C 180,E1 7658.156,E2 7658.156} C_VEL
LIN {X 0,Y 457.229,Z 563.28,A -85,B 0,C 180,E1 7663.358,E2 7663.358} C_VEL
LIN {X 0,Y 457.029,Z 563.28,A -85,B 0,C 180,E1 7669.281,E2 7669.281} C_VEL
LIN {X 0,Y 456.807,Z 563.28,A -85,B 0,C 180,E1 7675.433,E2 7675.433} C_VEL
LIN {X 0,Y 456.657,Z 563.28,A -85,B 0,C 180,E1 7681.92,E2 7681.92} C_VEL
LIN {X 0,Y 456.724,Z 563.28,A -85,B 0,C 180,E1 7688.886,E2 7688.886} C_VEL
LIN {X 0,Y 456.671,Z 563.28,A -85,B 0,C 180,E1 7693.942,E2 7693.942} C_VEL
LIN {X 0,Y 456.662,Z 563.28,A -85,B 0,C 180,E1 7699.467,E2 7699.467} C_VEL
LIN {X 0,Y 456.633,Z 563.28,A -85,B 0,C 180,E1 7705.819,E2 7705.819} C_VEL
LIN {X 0,Y 456.804,Z 563.28,A -85,B 0,C 180,E1 7712.451,E2 7712.451} C_VEL
LIN {X 0,Y 457.013,Z 563.28,A -85,B 0,C 180,E1 7718.701,E2 7718.701} C_VEL
LIN {X 0,Y 456.985,Z 563.28,A -85,B 0,C 180,E1 7724.681,E2 7724.681} C_VEL
LIN {X 0,Y 457.246,Z 563.28,A -85,B 0,C 180,E1 7730.5,E2 7730.5} C_VEL
LIN {X 0,Y 457.495,Z 563.28,A -85,B 0,C 180,E1 7736.216,E2 7736.216} C_VEL
LIN {X 0,Y 457.479,Z 563.28,A -85,B 0,C 180,E1 7741.888,E2 7741.888} C_VEL
LIN {X 0,Y 457.302,Z 563.28,A -85,B 0,C 180,E1 7748.127,E2 7748.127} C_VEL
LIN {X 0,Y 457.279,Z 563.28,A -85,B 0,C 180,E1 7753.354,E2 7753.354} C_VEL
LIN {X 0,Y 457.043,Z 563.28,A -85,B 0,C 180,E1 7759.277,E2 7759.277} C_VEL
LIN {X 0,Y 456.829,Z 563.28,A -85,B 0,C 180,E1 7765.428,E2 7765.428} C_VEL
LIN {X 0,Y 456.801,Z 563.28,A -85,B 0,C 180,E1 7771.905,E2 7771.905} C_VEL
LIN {X 0,Y 456.709,Z 563.28,A -85,B 0,C 180,E1 7778.883,E2 7778.883} C_VEL
LIN {X 0,Y 456.561,Z 563.28,A -85,B 0,C 180,E1 7786.044,E2 7786.044} C_VEL
LIN {X 0,Y 456.627,Z 563.333,A -85,B 0,C 180,E1 7789.238,E2 7789.238} C_VEL
LIN {X 0,Y 460.867,Z 572.63,A -85,B 0,C 180,E1 7789.873,E2 7789.873} C_VEL
LIN {X 0,Y 481.632,Z 612.998,A -85,B 0,C 180,E1 7792.732,E2 7792.732} C_VEL
LIN {X 0,Y 478.951,Z 656.235,A -85,B 0,C 180,E1 7794.17,E2 7794.17} C_VEL
LIN {X 0,Y 476.49,Z 683.237,A -85,B 0,C 180,E1 7795.543,E2 7795.543} C_VEL
LIN {X 0,Y 471.354,Z 699.056,A -85,B 0,C 180,E1 7796.26,E2 7796.26} C_VEL
LIN {X 0,Y 466.216,Z 714.16,A -85,B 0,C 180,E1 7797.102,E2 7797.102} C_VEL
LIN {X 0,Y 461.578,Z 748.502,A -85,B 0,C 180,E1 7800.263,E2 7800.263} C_VEL
LIN {X 0,Y 457.572,Z 777.859,A -85,B 0,C 180,E1 7803.842,E2 7803.842} C_VEL
LIN {X 0,Y 453.994,Z 805.228,A -85,B 0,C 180,E1 7808.297,E2 7808.297} C_VEL
LIN {X 0,Y 451.838,Z 824.525,A -85,B 0,C 180,E1 7812.507,E2 7812.507} C_VEL
LIN {X 0,Y 450.464,Z 840.728,A -85,B 0,C 180,E1 7817.423,E2 7817.423} C_VEL
LIN {X 0,Y 449.988,Z 851.247,A -85,B 0,C 180,E1 7822.29,E2 7822.29} C_VEL
LIN {X 0,Y 449.831,Z 855.943,A -85,B 0,C 180,E1 7826.152,E2 7826.152} C_VEL
LIN {X 0,Y 449.844,Z 857.5,A -85,B 0,C 180,E1 7829.999,E2 7829.999} C_VEL
LIN {X 0,Y 449.806,Z 855.944,A -85,B 0,C 180,E1 7833.846,E2 7833.846} C_VEL
LIN {X 0,Y 450.058,Z 849.208,A -85,B 0,C 180,E1 7838.854,E2 7838.854} C_VEL
LIN {X 0,Y 450.809,Z 836.984,A -85,B 0,C 180,E1 7843.91,E2 7843.91} C_VEL
LIN {X 0,Y 452.429,Z 818.842,A -85,B 0,C 180,E1 7848.854,E2 7848.854} C_VEL
LIN {X 0,Y 455.01,Z 796.997,A -85,B 0,C 180,E1 7853.192,E2 7853.192} C_VEL
LIN {X 0,Y 459.11,Z 766.542,A -85,B 0,C 180,E1 7857.662,E2 7857.662} C_VEL
LIN {X 0,Y 463.599,Z 733.531,A -85,B 0,C 180,E1 7861.234,E2 7861.234} C_VEL
LIN {X 0,Y 468.143,Z 698.743,A -85,B 0,C 180,E1 7864.017,E2 7864.017} C_VEL
LIN {X 0,Y 472.137,Z 660.688,A -85,B 0,C 180,E1 7866.176,E2 7866.176} C_VEL
LIN {X 0,Y 474.936,Z 624.66,A -85,B 0,C 180,E1 7867.513,E2 7867.513} C_VEL
LIN {X 0,Y 474.777,Z 615.279,A -85,B 0,C 180,E1 7867.82,E2 7867.82} C_VEL
LIN {X 0,Y 455.589,Z 577.212,A -85,B 0,C 180,E1 7870.592,E2 7870.592} C_VEL
LIN {X 0,Y 448.813,Z 564.504,A -85,B 0,C 180,E1 7871.596,E2 7871.596} C_VEL
LIN {X 0,Y 448.714,Z 563.28,A -85,B 0,C 180,E1 7871.775,E2 7871.775} C_VEL
LIN {X 0,Y 448.691,Z 563.28,A -85,B 0,C 180,E1 7877.733,E2 7877.733} C_VEL
LIN {X 0,Y 448.683,Z 563.28,A -85,B 0,C 180,E1 7883.818,E2 7883.818} C_VEL
LIN {X 0,Y 448.732,Z 563.28,A -85,B 0,C 180,E1 7889.71,E2 7889.71} C_VEL
LIN {X 0,Y 448.937,Z 563.28,A -85,B 0,C 180,E1 7896.215,E2 7896.215} C_VEL
LIN {X 0,Y 449.129,Z 563.28,A -85,B 0,C 180,E1 7902.401,E2 7902.401} C_VEL
LIN {X 0,Y 449.191,Z 563.28,A -85,B 0,C 180,E1 7908.374,E2 7908.374} C_VEL
LIN {X 0,Y 449.557,Z 563.28,A -85,B 0,C 180,E1 7914.223,E2 7914.223} C_VEL
LIN {X 0,Y 449.704,Z 563.28,A -85,B 0,C 180,E1 7920.002,E2 7920.002} C_VEL
LIN {X 0,Y 449.521,Z 563.28,A -85,B 0,C 180,E1 7925.782,E2 7925.782} C_VEL
LIN {X 0,Y 449.312,Z 563.28,A -85,B 0,C 180,E1 7931.627,E2 7931.627} C_VEL
LIN {X 0,Y 449.165,Z 563.28,A -85,B 0,C 180,E1 7937.601,E2 7937.601} C_VEL
LIN {X 0,Y 448.96,Z 563.28,A -85,B 0,C 180,E1 7943.789,E2 7943.789} C_VEL
LIN {X 0,Y 448.854,Z 563.28,A -85,B 0,C 180,E1 7950.286,E2 7950.286} C_VEL
LIN {X 0,Y 448.831,Z 563.28,A -85,B 0,C 180,E1 7957.243,E2 7957.243} C_VEL
LIN {X 0,Y 448.663,Z 563.28,A -85,B 0,C 180,E1 7962.275,E2 7962.275} C_VEL
LIN {X 0,Y 448.664,Z 563.28,A -85,B 0,C 180,E1 7967.728,E2 7967.728} C_VEL
LIN {X 0,Y 448.83,Z 563.28,A -85,B 0,C 180,E1 7973.797,E2 7973.797} C_VEL
LIN {X 0,Y 448.873,Z 563.28,A -85,B 0,C 180,E1 7979.718,E2 7979.718} C_VEL
LIN {X 0,Y 448.899,Z 563.28,A -85,B 0,C 180,E1 7986.211,E2 7986.211} C_VEL
LIN {X 0,Y 449.134,Z 563.28,A -85,B 0,C 180,E1 7992.4,E2 7992.4} C_VEL
LIN {X 0,Y 449.354,Z 563.28,A -85,B 0,C 180,E1 7998.377,E2 7998.377} C_VEL
LIN {X 0,Y 449.539,Z 563.28,A -85,B 0,C 180,E1 8004.221,E2 8004.221} C_VEL
LIN {X 0,Y 449.715,Z 563.28,A -85,B 0,C 180,E1 8010.001,E2 8010.001} C_VEL
LIN {X 0,Y 449.599,Z 563.28,A -85,B 0,C 180,E1 8015.78,E2 8015.78} C_VEL
LIN {X 0,Y 449.295,Z 563.28,A -85,B 0,C 180,E1 8021.627,E2 8021.627} C_VEL
LIN {X 0,Y 449.124,Z 563.28,A -85,B 0,C 180,E1 8027.602,E2 8027.602} C_VEL
LIN {X 0,Y 448.939,Z 563.28,A -85,B 0,C 180,E1 8033.789,E2 8033.789} C_VEL
LIN {X 0,Y 448.722,Z 563.28,A -85,B 0,C 180,E1 8040.295,E2 8040.295} C_VEL
LIN {X 0,Y 448.795,Z 563.28,A -85,B 0,C 180,E1 8047.246,E2 8047.246} C_VEL
LIN {X 0,Y 448.723,Z 563.28,A -85,B 0,C 180,E1 8052.28,E2 8052.28} C_VEL
LIN {X 0,Y 448.723,Z 563.28,A -85,B 0,C 180,E1 8057.732,E2 8057.732} C_VEL
LIN {X 0,Y 448.685,Z 563.28,A -85,B 0,C 180,E1 8063.821,E2 8063.821} C_VEL
LIN {X 0,Y 448.735,Z 563.28,A -85,B 0,C 180,E1 8069.705,E2 8069.705} C_VEL
LIN {X 0,Y 448.962,Z 563.28,A -85,B 0,C 180,E1 8076.211,E2 8076.211} C_VEL
LIN {X 0,Y 449.146,Z 563.28,A -85,B 0,C 180,E1 8082.398,E2 8082.398} C_VEL
LIN {X 0,Y 449.187,Z 563.28,A -85,B 0,C 180,E1 8088.37,E2 8088.37} C_VEL
LIN {X 0,Y 449.57,Z 563.28,A -85,B 0,C 180,E1 8094.219,E2 8094.219} C_VEL
LIN {X 0,Y 449.715,Z 563.28,A -85,B 0,C 180,E1 8099.998,E2 8099.998} C_VEL
LIN {X 0,Y 449.529,Z 563.28,A -85,B 0,C 180,E1 8105.778,E2 8105.778} C_VEL
LIN {X 0,Y 449.353,Z 563.28,A -85,B 0,C 180,E1 8111.622,E2 8111.622} C_VEL
LIN {X 0,Y 449.142,Z 563.28,A -85,B 0,C 180,E1 8117.598,E2 8117.598} C_VEL
LIN {X 0,Y 448.945,Z 563.28,A -85,B 0,C 180,E1 8123.785,E2 8123.785} C_VEL
LIN {X 0,Y 448.852,Z 563.28,A -85,B 0,C 180,E1 8130.281,E2 8130.281} C_VEL
LIN {X 0,Y 448.816,Z 563.28,A -85,B 0,C 180,E1 8137.24,E2 8137.24} C_VEL
LIN {X 0,Y 448.652,Z 563.28,A -85,B 0,C 180,E1 8142.271,E2 8142.271} C_VEL
LIN {X 0,Y 448.684,Z 563.28,A -85,B 0,C 180,E1 8148.336,E2 8148.336} C_VEL
LIN {X 0,Y 453.392,Z 573.365,A -85,B 0,C 180,E1 8149.093,E2 8149.093} C_VEL
LIN {X 0,Y 473.704,Z 612.273,A -85,B 0,C 180,E1 8151.986,E2 8151.986} C_VEL
LIN {X 0,Y 475.223,Z 618.297,A -85,B 0,C 180,E1 8152.315,E2 8152.315} C_VEL
LIN {X 0,Y 472.375,Z 657.555,A -85,B 0,C 180,E1 8153.669,E2 8153.669} C_VEL
LIN {X 0,Y 468.261,Z 696.846,A -85,B 0,C 180,E1 8155.851,E2 8155.851} C_VEL
LIN {X 0,Y 466.216,Z 714.16,A -85,B 0,C 180,E1 8157.102,E2 8157.102} C_VEL
LIN {X 0,Y 460.836,Z 728.977,A -85,B 0,C 180,E1 8158.064,E2 8158.064} C_VEL
LIN {X 0,Y 455.645,Z 741.287,A -85,B 0,C 180,E1 8159.014,E2 8159.014} C_VEL
LIN {X 0,Y 455.319,Z 742.963,A -85,B 0,C 180,E1 8159.186,E2 8159.186} C_VEL
LIN {X 0,Y 450.406,Z 776.491,A -85,B 0,C 180,E1 8163.225,E2 8163.225} C_VEL
LIN {X 0,Y 446.651,Z 803.62,A -85,B 0,C 180,E1 8167.66,E2 8167.66} C_VEL
LIN {X 0,Y 444.114,Z 824.467,A -85,B 0,C 180,E1 8172.193,E2 8172.193} C_VEL
LIN {X 0,Y 442.649,Z 840.725,A -85,B 0,C 180,E1 8177.197,E2 8177.197} C_VEL
LIN {X 0,Y 442.124,Z 850.694,A -85,B 0,C 180,E1 8181.787,E2 8181.787} C_VEL
LIN {X 0,Y 441.924,Z 855.939,A -85,B 0,C 180,E1 8186.083,E2 8186.083} C_VEL
LIN {X 0,Y 441.944,Z 857.5,A -85,B 0,C 180,E1 8189.999,E2 8189.999} C_VEL
LIN {X 0,Y 441.902,Z 855.94,A -85,B 0,C 180,E1 8193.915,E2 8193.915} C_VEL
LIN {X 0,Y 442.18,Z 849.45,A -85,B 0,C 180,E1 8198.882,E2 8198.882} C_VEL
LIN {X 0,Y 442.985,Z 836.984,A -85,B 0,C 180,E1 8204.16,E2 8204.16} C_VEL
LIN {X 0,Y 444.568,Z 820.215,A -85,B 0,C 180,E1 8208.836,E2 8208.836} C_VEL
LIN {X 0,Y 447.304,Z 798.201,A -85,B 0,C 180,E1 8213.352,E2 8213.352} C_VEL
LIN {X 0,Y 451.329,Z 769.77,A -85,B 0,C 180,E1 8217.678,E2 8217.678} C_VEL
LIN {X 0,Y 455.976,Z 738.562,A -85,B 0,C 180,E1 8221.252,E2 8221.252} C_VEL
LIN {X 0,Y 460.912,Z 702.963,A -85,B 0,C 180,E1 8224.267,E2 8224.267} C_VEL
LIN {X 0,Y 465.115,Z 666.255,A -85,B 0,C 180,E1 8226.473,E2 8226.473} C_VEL
LIN {X 0,Y 468.338,Z 629.089,A -85,B 0,C 180,E1 8227.966,E2 8227.966} C_VEL
LIN {X 0,Y 468.445,Z 618.119,A -85,B 0,C 180,E1 8228.325,E2 8228.325} C_VEL
LIN {X 0,Y 450.325,Z 581.762,A -85,B 0,C 180,E1 8231.069,E2 8231.069} C_VEL
LIN {X 0,Y 440.853,Z 564.482,A -85,B 0,C 180,E1 8232.514,E2 8232.514} C_VEL
LIN {X 0,Y 440.759,Z 563.28,A -85,B 0,C 180,E1 8232.636,E2 8232.636} C_VEL
LIN {X 0,Y 440.705,Z 563.28,A -85,B 0,C 180,E1 8239.418,E2 8239.418} C_VEL
LIN {X 0,Y 440.763,Z 563.28,A -85,B 0,C 180,E1 8245.251,E2 8245.251} C_VEL
LIN {X 0,Y 440.879,Z 563.28,A -85,B 0,C 180,E1 8251.371,E2 8251.371} C_VEL
LIN {X 0,Y 441.088,Z 563.28,A -85,B 0,C 180,E1 8257.897,E2 8257.897} C_VEL
LIN {X 0,Y 441.155,Z 563.28,A -85,B 0,C 180,E1 8264.121,E2 8264.121} C_VEL
LIN {X 0,Y 441.378,Z 563.28,A -85,B 0,C 180,E1 8270.16,E2 8270.16} C_VEL
LIN {X 0,Y 441.661,Z 563.28,A -85,B 0,C 180,E1 8276.084,E2 8276.084} C_VEL
LIN {X 0,Y 441.737,Z 563.28,A -85,B 0,C 180,E1 8281.96,E2 8281.96} C_VEL
LIN {X 0,Y 441.533,Z 563.28,A -85,B 0,C 180,E1 8287.859,E2 8287.859} C_VEL
LIN {X 0,Y 441.407,Z 563.28,A -85,B 0,C 180,E1 8293.847,E2 8293.847} C_VEL
LIN {X 0,Y 441.183,Z 563.28,A -85,B 0,C 180,E1 8300.003,E2 8300.003} C_VEL
LIN {X 0,Y 440.962,Z 563.28,A -85,B 0,C 180,E1 8306.417,E2 8306.417} C_VEL
LIN {X 0,Y 440.895,Z 563.28,A -85,B 0,C 180,E1 8313.206,E2 8313.206} C_VEL
LIN {X 0,Y 440.841,Z 563.28,A -85,B 0,C 180,E1 8318.068,E2 8318.068} C_VEL
LIN {X 0,Y 440.634,Z 563.28,A -85,B 0,C 180,E1 8324.015,E2 8324.015} C_VEL
LIN {X 0,Y 440.728,Z 563.28,A -85,B 0,C 180,E1 8329.419,E2 8329.419} C_VEL
LIN {X 0,Y 440.924,Z 563.28,A -85,B 0,C 180,E1 8335.225,E2 8335.225} C_VEL
LIN {X 0,Y 440.959,Z 563.28,A -85,B 0,C 180,E1 8341.375,E2 8341.375} C_VEL
LIN {X 0,Y 441.033,Z 563.28,A -85,B 0,C 180,E1 8347.892,E2 8347.892} C_VEL
LIN {X 0,Y 441.303,Z 563.28,A -85,B 0,C 180,E1 8354.125,E2 8354.125} C_VEL
LIN {X 0,Y 441.521,Z 563.28,A -85,B 0,C 180,E1 8360.161,E2 8360.161} C_VEL
LIN {X 0,Y 441.75,Z 563.28,A -85,B 0,C 180,E1 8366.083,E2 8366.083} C_VEL
LIN {X 0,Y 441.914,Z 563.28,A -85,B 0,C 180,E1 8371.958,E2 8371.958} C_VEL
LIN {X 0,Y 441.564,Z 563.28,A -85,B 0,C 180,E1 8377.858,E2 8377.858} C_VEL
LIN {X 0,Y 441.349,Z 563.28,A -85,B 0,C 180,E1 8383.848,E2 8383.848} C_VEL
LIN {X 0,Y 441.155,Z 563.28,A -85,B 0,C 180,E1 8390.003,E2 8390.003} C_VEL
LIN {X 0,Y 440.907,Z 563.28,A -85,B 0,C 180,E1 8396.42,E2 8396.42} C_VEL
LIN {X 0,Y 440.757,Z 563.28,A -85,B 0,C 180,E1 8403.217,E2 8403.217} C_VEL
LIN {X 0,Y 440.836,Z 563.28,A -85,B 0,C 180,E1 8408.064,E2 8408.064} C_VEL
LIN {X 0,Y 440.708,Z 563.28,A -85,B 0,C 180,E1 8414.022,E2 8414.022} C_VEL
LIN {X 0,Y 440.732,Z 563.28,A -85,B 0,C 180,E1 8419.416,E2 8419.416} C_VEL
LIN {X 0,Y 440.771,Z 563.28,A -85,B 0,C 180,E1 8425.253,E2 8425.253} C_VEL
LIN {X 0,Y 440.89,Z 563.28,A -85,B 0,C 180,E1 8431.367,E2 8431.367} C_VEL
LIN {X 0,Y 441.107,Z 563.28,A -85,B 0,C 180,E1 8437.893,E2 8437.893} C_VEL
LIN {X 0,Y 441.163,Z 563.28,A -85,B 0,C 180,E1 8444.117,E2 8444.117} C_VEL
LIN {X 0,Y 441.394,Z 563.28,A -85,B 0,C 180,E1 8450.156,E2 8450.156} C_VEL
LIN {X 0,Y 441.675,Z 563.28,A -85,B 0,C 180,E1 8456.08,E2 8456.08} C_VEL
LIN {X 0,Y 441.694,Z 563.28,A -85,B 0,C 180,E1 8461.956,E2 8461.956} C_VEL
LIN {X 0,Y 441.542,Z 563.28,A -85,B 0,C 180,E1 8467.855,E2 8467.855} C_VEL
LIN {X 0,Y 441.413,Z 563.28,A -85,B 0,C 180,E1 8473.843,E2 8473.843} C_VEL
LIN {X 0,Y 441.167,Z 563.28,A -85,B 0,C 180,E1 8479.999,E2 8479.999} C_VEL
LIN {X 0,Y 440.946,Z 563.28,A -85,B 0,C 180,E1 8486.413,E2 8486.413} C_VEL
LIN {X 0,Y 440.894,Z 563.28,A -85,B 0,C 180,E1 8493.201,E2 8493.201} C_VEL
LIN {X 0,Y 440.823,Z 563.28,A -85,B 0,C 180,E1 8498.062,E2 8498.062} C_VEL
LIN {X 0,Y 440.613,Z 563.28,A -85,B 0,C 180,E1 8504.01,E2 8504.01} C_VEL
LIN {X 0,Y 440.697,Z 563.28,A -85,B 0,C 180,E1 8507.429,E2 8507.429} C_VEL
LIN {X 0,Y 443.311,Z 569.094,A -85,B 0,C 180,E1 8507.872,E2 8507.872} C_VEL
LIN {X 0,Y 465.809,Z 611.718,A -85,B 0,C 180,E1 8511.215,E2 8511.215} C_VEL
LIN {X 0,Y 468.871,Z 618.642,A -85,B 0,C 180,E1 8511.732,E2 8511.732} C_VEL
LIN {X 0,Y 465.817,Z 658.637,A -85,B 0,C 180,E1 8513.149,E2 8513.149} C_VEL
LIN {X 0,Y 461.375,Z 698.69,A -85,B 0,C 180,E1 8515.429,E2 8515.429} C_VEL
LIN {X 0,Y 456.601,Z 734.074,A -85,B 0,C 180,E1 8518.317,E2 8518.317} C_VEL
LIN {X 0,Y 455.319,Z 742.963,A -85,B 0,C 180,E1 8519.186,E2 8519.186} C_VEL
LIN {X 0,Y 449.806,Z 756.476,A -85,B 0,C 180,E1 8520.435,E2 8520.435} C_VEL
LIN {X 0,Y 444.173,Z 769.205,A -85,B 0,C 180,E1 8521.791,E2 8521.791} C_VEL
LIN {X 0,Y 439.902,Z 797.94,A -85,B 0,C 180,E1 8526.229,E2 8526.229} C_VEL
LIN {X 0,Y 436.655,Z 822.203,A -85,B 0,C 180,E1 8531.356,E2 8531.356} C_VEL
LIN {X 0,Y 434.99,Z 838.696,A -85,B 0,C 180,E1 8536.237,E2 8536.237} C_VEL
LIN {X 0,Y 434.292,Z 849.537,A -85,B 0,C 180,E1 8541.003,E2 8541.003} C_VEL
LIN {X 0,Y 434.039,Z 855.936,A -85,B 0,C 180,E1 8546.012,E2 8546.012} C_VEL
LIN {X 0,Y 434.044,Z 857.5,A -85,B 0,C 180,E1 8549.999,E2 8549.999} C_VEL
LIN {X 0,Y 434.021,Z 855.937,A -85,B 0,C 180,E1 8553.986,E2 8553.986} C_VEL
LIN {X 0,Y 434.286,Z 849.54,A -85,B 0,C 180,E1 8558.995,E2 8558.995} C_VEL
LIN {X 0,Y 435.087,Z 837.907,A -85,B 0,C 180,E1 8564.05,E2 8564.05} C_VEL
LIN {X 0,Y 436.729,Z 821.139,A -85,B 0,C 180,E1 8568.9,E2 8568.9} C_VEL
LIN {X 0,Y 439.833,Z 797.948,A -85,B 0,C 180,E1 8573.773,E2 8573.773} C_VEL
LIN {X 0,Y 444.162,Z 769.21,A -85,B 0,C 180,E1 8578.209,E2 8578.209} C_VEL
LIN {X 0,Y 449.037,Z 738.089,A -85,B 0,C 180,E1 8581.814,E2 8581.814} C_VEL
LIN {X 0,Y 454.472,Z 701.367,A -85,B 0,C 180,E1 8584.94,E2 8584.94} C_VEL
LIN {X 0,Y 458.963,Z 663.67,A -85,B 0,C 180,E1 8587.182,E2 8587.182} C_VEL
LIN {X 0,Y 462.304,Z 626.74,A -85,B 0,C 180,E1 8588.638,E2 8588.638} C_VEL
LIN {X 0,Y 461.758,Z 620.172,A -85,B 0,C 180,E1 8588.908,E2 8588.908} C_VEL
LIN {X 0,Y 444.165,Z 584.537,A -85,B 0,C 180,E1 8591.702,E2 8591.702} C_VEL
LIN {X 0,Y 432.946,Z 564.752,A -85,B 0,C 180,E1 8593.468,E2 8593.468} C_VEL
LIN {X 0,Y 432.804,Z 563.28,A -85,B 0,C 180,E1 8593.618,E2 8593.618} C_VEL
LIN {X 0,Y 432.735,Z 563.28,A -85,B 0,C 180,E1 8600.099,E2 8600.099} C_VEL
LIN {X 0,Y 432.817,Z 563.28,A -85,B 0,C 180,E1 8606.797,E2 8606.797} C_VEL
LIN {X 0,Y 432.992,Z 563.28,A -85,B 0,C 180,E1 8613.063,E2 8613.063} C_VEL
LIN {X 0,Y 433.289,Z 563.28,A -85,B 0,C 180,E1 8620.103,E2 8620.103} C_VEL
LIN {X 0,Y 433.273,Z 563.28,A -85,B 0,C 180,E1 8625.892,E2 8625.892} C_VEL
LIN {X 0,Y 433.606,Z 563.28,A -85,B 0,C 180,E1 8632,E2 8632} C_VEL
LIN {X 0,Y 433.984,Z 563.28,A -85,B 0,C 180,E1 8638.009,E2 8638.009} C_VEL
LIN {X 0,Y 433.824,Z 563.28,A -85,B 0,C 180,E1 8643.991,E2 8643.991} C_VEL
LIN {X 0,Y 433.546,Z 563.28,A -85,B 0,C 180,E1 8650.024,E2 8650.024} C_VEL
LIN {X 0,Y 433.388,Z 563.28,A -85,B 0,C 180,E1 8656.176,E2 8656.176} C_VEL
LIN {X 0,Y 433.189,Z 563.28,A -85,B 0,C 180,E1 8662.533,E2 8662.533} C_VEL
LIN {X 0,Y 432.97,Z 563.28,A -85,B 0,C 180,E1 8669.39,E2 8669.39} C_VEL
LIN {X 0,Y 432.991,Z 563.28,A -85,B 0,C 180,E1 8673.893,E2 8673.893} C_VEL
LIN {X 0,Y 432.775,Z 563.28,A -85,B 0,C 180,E1 8679.907,E2 8679.907} C_VEL
LIN {X 0,Y 432.709,Z 563.28,A -85,B 0,C 180,E1 8687.085,E2 8687.085} C_VEL
LIN {X 0,Y 432.902,Z 563.28,A -85,B 0,C 180,E1 8693.66,E2 8693.66} C_VEL
LIN {X 0,Y 432.976,Z 563.28,A -85,B 0,C 180,E1 8698.482,E2 8698.482} C_VEL
LIN {X 0,Y 433.009,Z 563.28,A -85,B 0,C 180,E1 8705.281,E2 8705.281} C_VEL
LIN {X 0,Y 433.255,Z 563.28,A -85,B 0,C 180,E1 8711.733,E2 8711.733} C_VEL
LIN {X 0,Y 433.518,Z 563.28,A -85,B 0,C 180,E1 8717.946,E2 8717.946} C_VEL
LIN {X 0,Y 433.72,Z 563.28,A -85,B 0,C 180,E1 8724.01,E2 8724.01} C_VEL
LIN {X 0,Y 433.913,Z 563.28,A -85,B 0,C 180,E1 8730.001,E2 8730.001} C_VEL
LIN {X 0,Y 433.772,Z 563.28,A -85,B 0,C 180,E1 8735.991,E2 8735.991} C_VEL
LIN {X 0,Y 433.406,Z 563.28,A -85,B 0,C 180,E1 8742.862,E2 8742.862} C_VEL
LIN {X 0,Y 433.258,Z 563.28,A -85,B 0,C 180,E1 8748.269,E2 8748.269} C_VEL
LIN {X 0,Y 432.996,Z 563.28,A -85,B 0,C 180,E1 8755.024,E2 8755.024} C_VEL
LIN {X 0,Y 432.794,Z 563.28,A -85,B 0,C 180,E1 8761.535,E2 8761.535} C_VEL
LIN {X 0,Y 432.863,Z 563.28,A -85,B 0,C 180,E1 8766.695,E2 8766.695} C_VEL
LIN {X 0,Y 432.83,Z 563.28,A -85,B 0,C 180,E1 8772.932,E2 8772.932} C_VEL
LIN {X 0,Y 432.803,Z 563.28,A -85,B 0,C 180,E1 8778.511,E2 8778.511} C_VEL
LIN {X 0,Y 432.792,Z 563.28,A -85,B 0,C 180,E1 8783.647,E2 8783.647} C_VEL
LIN {X 0,Y 432.871,Z 563.28,A -85,B 0,C 180,E1 8790.637,E2 8790.637} C_VEL
LIN {X 0,Y 433.168,Z 563.28,A -85,B 0,C 180,E1 8797.466,E2 8797.466} C_VEL
LIN {X 0,Y 433.269,Z 563.28,A -85,B 0,C 180,E1 8803.82,E2 8803.82} C_VEL
LIN {X 0,Y 433.458,Z 563.28,A -85,B 0,C 180,E1 8809.974,E2 8809.974} C_VEL
LIN {X 0,Y 433.77,Z 563.28,A -85,B 0,C 180,E1 8816.008,E2 8816.008} C_VEL
LIN {X 0,Y 433.79,Z 563.28,A -85,B 0,C 180,E1 8821.991,E2 8821.991} C_VEL
LIN {X 0,Y 433.621,Z 563.28,A -85,B 0,C 180,E1 8827.999,E2 8827.999} C_VEL
LIN {X 0,Y 433.468,Z 563.28,A -85,B 0,C 180,E1 8834.102,E2 8834.102} C_VEL
LIN {X 0,Y 433.232,Z 563.28,A -85,B 0,C 180,E1 8840.382,E2 8840.382} C_VEL
LIN {X 0,Y 433.026,Z 563.28,A -85,B 0,C 180,E1 8846.935,E2 8846.935} C_VEL
LIN {X 0,Y 432.989,Z 563.28,A -85,B 0,C 180,E1 8853.888,E2 8853.888} C_VEL
LIN {X 0,Y 432.757,Z 563.28,A -85,B 0,C 180,E1 8859.901,E2 8859.901} C_VEL
LIN {X 0,Y 432.71,Z 563.34,A -85,B 0,C 180,E1 8866.471,E2 8866.471} C_VEL
LIN {X 0,Y 435.281,Z 569.063,A -85,B 0,C 180,E1 8866.916,E2 8866.916} C_VEL
LIN {X 0,Y 457.225,Z 609.643,A -85,B 0,C 180,E1 8870.297,E2 8870.297} C_VEL
LIN {X 0,Y 462.481,Z 622.427,A -85,B 0,C 180,E1 8871.236,E2 8871.236} C_VEL
LIN {X 0,Y 459.165,Z 661.147,A -85,B 0,C 180,E1 8872.688,E2 8872.688} C_VEL
LIN {X 0,Y 454.58,Z 700.019,A -85,B 0,C 180,E1 8874.96,E2 8874.96} C_VEL
LIN {X 0,Y 449.46,Z 735.471,A -85,B 0,C 180,E1 8877.934,E2 8877.934} C_VEL
LIN {X 0,Y 444.721,Z 766.021,A -85,B 0,C 180,E1 8881.36,E2 8881.36} C_VEL
LIN {X 0,Y 444.173,Z 769.205,A -85,B 0,C 180,E1 8881.791,E2 8881.791} C_VEL
LIN {X 0,Y 438.613,Z 781.295,A -85,B 0,C 180,E1 8883.286,E2 8883.286} C_VEL
LIN {X 0,Y 433.164,Z 792.539,A -85,B 0,C 180,E1 8884.894,E2 8884.894} C_VEL
LIN {X 0,Y 429.746,Z 815.524,A -85,B 0,C 180,E1 8889.442,E2 8889.442} C_VEL
LIN {X 0,Y 427.558,Z 834.581,A -85,B 0,C 180,E1 8894.65,E2 8894.65} C_VEL
LIN {X 0,Y 426.584,Z 847.532,A -85,B 0,C 180,E1 8899.811,E2 8899.811} C_VEL
LIN {X 0,Y 426.185,Z 853.957,A -85,B 0,C 180,E1 8903.901,E2 8903.901} C_VEL
LIN {X 0,Y 426.125,Z 857.106,A -85,B 0,C 180,E1 8907.97,E2 8907.97} C_VEL
LIN {X 0,Y 426.159,Z 857.106,A -85,B 0,C 180,E1 8912.028,E2 8912.028} C_VEL
LIN {X 0,Y 426.296,Z 852.958,A -85,B 0,C 180,E1 8916.884,E2 8916.884} C_VEL
LIN {X 0,Y 426.808,Z 843.044,A -85,B 0,C 180,E1 8922.246,E2 8922.246} C_VEL
LIN {X 0,Y 428.243,Z 828.414,A -85,B 0,C 180,E1 8927.237,E2 8927.237} C_VEL
LIN {X 0,Y 430.941,Z 807.655,A -85,B 0,C 180,E1 8932.263,E2 8932.263} C_VEL
LIN {X 0,Y 434.858,Z 782.07,A -85,B 0,C 180,E1 8936.814,E2 8936.814} C_VEL
LIN {X 0,Y 439.747,Z 752.372,A -85,B 0,C 180,E1 8940.805,E2 8940.805} C_VEL
LIN {X 0,Y 445.534,Z 716.643,A -85,B 0,C 180,E1 8944.322,E2 8944.322} C_VEL
LIN {X 0,Y 450.52,Z 679.976,A -85,B 0,C 180,E1 8946.914,E2 8946.914} C_VEL
LIN {X 0,Y 454.852,Z 640.654,A -85,B 0,C 180,E1 8948.793,E2 8948.793} C_VEL
LIN {X 0,Y 455.72,Z 623.582,A -85,B 0,C 180,E1 8949.402,E2 8949.402} C_VEL
LIN {X 0,Y 439.09,Z 589.409,A -85,B 0,C 180,E1 8952.185,E2 8952.185} C_VEL
LIN {X 0,Y 424.951,Z 564.334,A -85,B 0,C 180,E1 8954.5,E2 8954.5} C_VEL
LIN {X 0,Y 424.871,Z 563.28,A -85,B 0,C 180,E1 8954.742,E2 8954.742} C_VEL
LIN {X 0,Y 424.842,Z 563.28,A -85,B 0,C 180,E1 8961.39,E2 8961.39} C_VEL
LIN {X 0,Y 424.89,Z 563.28,A -85,B 0,C 180,E1 8968.468,E2 8968.468} C_VEL
LIN {X 0,Y 425.095,Z 563.28,A -85,B 0,C 180,E1 8974.79,E2 8974.79} C_VEL
LIN {X 0,Y 425.345,Z 563.28,A -85,B 0,C 180,E1 8981.382,E2 8981.382} C_VEL
LIN {X 0,Y 425.442,Z 563.28,A -85,B 0,C 180,E1 8987.715,E2 8987.715} C_VEL
LIN {X 0,Y 425.81,Z 563.28,A -85,B 0,C 180,E1 8993.899,E2 8993.899} C_VEL
LIN {X 0,Y 426.002,Z 563.28,A -85,B 0,C 180,E1 9000.002,E2 9000.002} C_VEL
LIN {X 0,Y 425.779,Z 563.28,A -85,B 0,C 180,E1 9006.105,E2 9006.105} C_VEL
LIN {X 0,Y 425.59,Z 563.28,A -85,B 0,C 180,E1 9012.285,E2 9012.285} C_VEL
LIN {X 0,Y 425.365,Z 563.28,A -85,B 0,C 180,E1 9018.621,E2 9018.621} C_VEL
LIN {X 0,Y 425.134,Z 563.28,A -85,B 0,C 180,E1 9025.212,E2 9025.212} C_VEL
LIN {X 0,Y 425.035,Z 563.28,A -85,B 0,C 180,E1 9032.18,E2 9032.18} C_VEL
LIN {X 0,Y 424.914,Z 563.28,A -85,B 0,C 180,E1 9038.622,E2 9038.622} C_VEL
LIN {X 0,Y 424.777,Z 563.28,A -85,B 0,C 180,E1 9045.277,E2 9045.277} C_VEL
LIN {X 0,Y 424.915,Z 563.28,A -85,B 0,C 180,E1 9051.381,E2 9051.381} C_VEL
LIN {X 0,Y 425.076,Z 563.28,A -85,B 0,C 180,E1 9058.432,E2 9058.432} C_VEL
LIN {X 0,Y 425.087,Z 563.28,A -85,B 0,C 180,E1 9064.788,E2 9064.788} C_VEL
LIN {X 0,Y 425.317,Z 563.28,A -85,B 0,C 180,E1 9071.379,E2 9071.379} C_VEL
LIN {X 0,Y 425.619,Z 563.28,A -85,B 0,C 180,E1 9077.719,E2 9077.719} C_VEL
LIN {X 0,Y 425.8,Z 563.28,A -85,B 0,C 180,E1 9083.898,E2 9083.898} C_VEL
LIN {X 0,Y 426.012,Z 563.28,A -85,B 0,C 180,E1 9090.001,E2 9090.001} C_VEL
LIN {X 0,Y 425.849,Z 563.28,A -85,B 0,C 180,E1 9096.103,E2 9096.103} C_VEL
LIN {X 0,Y 425.556,Z 563.28,A -85,B 0,C 180,E1 9102.285,E2 9102.285} C_VEL
LIN {X 0,Y 425.332,Z 563.28,A -85,B 0,C 180,E1 9108.622,E2 9108.622} C_VEL
LIN {X 0,Y 425.091,Z 563.28,A -85,B 0,C 180,E1 9115.214,E2 9115.214} C_VEL
LIN {X 0,Y 424.899,Z 563.28,A -85,B 0,C 180,E1 9122.19,E2 9122.19} C_VEL
LIN {X 0,Y 424.913,Z 563.28,A -85,B 0,C 180,E1 9128.619,E2 9128.619} C_VEL
LIN {X 0,Y 424.903,Z 563.28,A -85,B 0,C 180,E1 9135.259,E2 9135.259} C_VEL
LIN {X 0,Y 424.87,Z 563.28,A -85,B 0,C 180,E1 9141.388,E2 9141.388} C_VEL
LIN {X 0,Y 424.905,Z 563.28,A -85,B 0,C 180,E1 9148.469,E2 9148.469} C_VEL
LIN {X 0,Y 425.115,Z 563.28,A -85,B 0,C 180,E1 9154.787,E2 9154.787} C_VEL
LIN {X 0,Y 425.364,Z 563.28,A -85,B 0,C 180,E1 9161.379,E2 9161.379} C_VEL
LIN {X 0,Y 425.413,Z 563.28,A -85,B 0,C 180,E1 9167.71,E2 9167.71} C_VEL
LIN {X 0,Y 425.823,Z 563.28,A -85,B 0,C 180,E1 9173.895,E2 9173.895} C_VEL
LIN {X 0,Y 426.011,Z 563.28,A -85,B 0,C 180,E1 9179.998,E2 9179.998} C_VEL
LIN {X 0,Y 425.789,Z 563.28,A -85,B 0,C 180,E1 9186.101,E2 9186.101} C_VEL
LIN {X 0,Y 425.619,Z 563.28,A -85,B 0,C 180,E1 9192.28,E2 9192.28} C_VEL
LIN {X 0,Y 425.345,Z 563.28,A -85,B 0,C 180,E1 9198.618,E2 9198.618} C_VEL
LIN {X 0,Y 425.113,Z 563.28,A -85,B 0,C 180,E1 9205.209,E2 9205.209} C_VEL
LIN {X 0,Y 425.034,Z 563.28,A -85,B 0,C 180,E1 9212.175,E2 9212.175} C_VEL
LIN {X 0,Y 424.897,Z 563.28,A -85,B 0,C 180,E1 9218.617,E2 9218.617} C_VEL
LIN {X 0,Y 424.801,Z 563.733,A -85,B 0,C 180,E1 9225.466,E2 9225.466} C_VEL
LIN {X 0,Y 429.791,Z 573.571,A -85,B 0,C 180,E1 9226.334,E2 9226.334} C_VEL
LIN {X 0,Y 450.106,Z 610.512,A -85,B 0,C 180,E1 9229.572,E2 9229.572} C_VEL
LIN {X 0,Y 456.142,Z 625.076,A -85,B 0,C 180,E1 9230.69,E2 9230.69} C_VEL
LIN {X 0,Y 452.388,Z 664.767,A -85,B 0,C 180,E1 9232.266,E2 9232.266} C_VEL
LIN {X 0,Y 447.584,Z 702.433,A -85,B 0,C 180,E1 9234.56,E2 9234.56} C_VEL
LIN {X 0,Y 441.971,Z 739.125,A -85,B 0,C 180,E1 9237.759,E2 9237.759} C_VEL
LIN {X 0,Y 436.761,Z 770.374,A -85,B 0,C 180,E1 9241.481,E2 9241.481} C_VEL
LIN {X 0,Y 433.164,Z 792.539,A -85,B 0,C 180,E1 9244.894,E2 9244.894} C_VEL
LIN {X 0,Y 427.693,Z 803.053,A -85,B 0,C 180,E1 9246.627,E2 9246.627} C_VEL
LIN {X 0,Y 422.485,Z 812.673,A -85,B 0,C 180,E1 9248.472,E2 9248.472} C_VEL
LIN {X 0,Y 420.04,Z 831.059,A -85,B 0,C 180,E1 9253.296,E2 9253.296} C_VEL
LIN {X 0,Y 418.804,Z 845.128,A -85,B 0,C 180,E1 9258.569,E2 9258.569} C_VEL
LIN {X 0,Y 418.326,Z 853.712,A -85,B 0,C 180,E1 9263.786,E2 9263.786} C_VEL
LIN {X 0,Y 418.238,Z 856.902,A -85,B 0,C 180,E1 9267.931,E2 9267.931} C_VEL
LIN {X 0,Y 418.269,Z 856.903,A -85,B 0,C 180,E1 9272.067,E2 9272.067} C_VEL
LIN {X 0,Y 418.408,Z 852,A -85,B 0,C 180,E1 9277.521,E2 9277.521} C_VEL
LIN {X 0,Y 419.097,Z 841.457,A -85,B 0,C 180,E1 9283.057,E2 9283.057} C_VEL
LIN {X 0,Y 420.794,Z 825.661,A -85,B 0,C 180,E1 9288.269,E2 9288.269} C_VEL
LIN {X 0,Y 423.675,Z 805.582,A -85,B 0,C 180,E1 9293.065,E2 9293.065} C_VEL
LIN {X 0,Y 428.337,Z 777.275,A -85,B 0,C 180,E1 9298.021,E2 9298.021} C_VEL
LIN {X 0,Y 433.888,Z 746.057,A -85,B 0,C 180,E1 9302.03,E2 9302.03} C_VEL
LIN {X 0,Y 439.444,Z 713.086,A -85,B 0,C 180,E1 9305.193,E2 9305.193} C_VEL
LIN {X 0,Y 444.99,Z 674.033,A -85,B 0,C 180,E1 9307.86,E2 9307.86} C_VEL
LIN {X 0,Y 449.065,Z 635.838,A -85,B 0,C 180,E1 9309.586,E2 9309.586} C_VEL
LIN {X 0,Y 449.304,Z 626.016,A -85,B 0,C 180,E1 9309.984,E2 9309.984} C_VEL
LIN {X 0,Y 433.261,Z 592.889,A -85,B 0,C 180,E1 9312.805,E2 9312.805} C_VEL
LIN {X 0,Y 417.074,Z 564.659,A -85,B 0,C 180,E1 9315.557,E2 9315.557} C_VEL
LIN {X 0,Y 416.944,Z 563.28,A -85,B 0,C 180,E1 9315.753,E2 9315.753} C_VEL
LIN {X 0,Y 416.98,Z 563.28,A -85,B 0,C 180,E1 9322.763,E2 9322.763} C_VEL
LIN {X 0,Y 417.014,Z 563.28,A -85,B 0,C 180,E1 9330.279,E2 9330.279} C_VEL
LIN {X 0,Y 417.215,Z 563.28,A -85,B 0,C 180,E1 9336.559,E2 9336.559} C_VEL
LIN {X 0,Y 417.413,Z 563.28,A -85,B 0,C 180,E1 9343.192,E2 9343.192} C_VEL
LIN {X 0,Y 417.579,Z 563.28,A -85,B 0,C 180,E1 9349.593,E2 9349.593} C_VEL
LIN {X 0,Y 417.933,Z 563.28,A -85,B 0,C 180,E1 9355.861,E2 9355.861} C_VEL
LIN {X 0,Y 418.052,Z 563.28,A -85,B 0,C 180,E1 9362.071,E2 9362.071} C_VEL
LIN {X 0,Y 417.762,Z 563.28,A -85,B 0,C 180,E1 9368.31,E2 9368.31} C_VEL
LIN {X 0,Y 417.592,Z 563.28,A -85,B 0,C 180,E1 9374.654,E2 9374.654} C_VEL
LIN {X 0,Y 417.354,Z 563.28,A -85,B 0,C 180,E1 9381.198,E2 9381.198} C_VEL
LIN {X 0,Y 417.104,Z 563.28,A -85,B 0,C 180,E1 9388.057,E2 9388.057} C_VEL
LIN {X 0,Y 417.054,Z 563.28,A -85,B 0,C 180,E1 9395.377,E2 9395.377} C_VEL
LIN {X 0,Y 416.916,Z 563.28,A -85,B 0,C 180,E1 9400.657,E2 9400.657} C_VEL
LIN {X 0,Y 416.814,Z 563.28,A -85,B 0,C 180,E1 9406.54,E2 9406.54} C_VEL
LIN {X 0,Y 417.071,Z 563.28,A -85,B 0,C 180,E1 9412.751,E2 9412.751} C_VEL
LIN {X 0,Y 417.121,Z 563.28,A -85,B 0,C 180,E1 9419.572,E2 9419.572} C_VEL
LIN {X 0,Y 417.193,Z 563.28,A -85,B 0,C 180,E1 9426.556,E2 9426.556} C_VEL
LIN {X 0,Y 417.487,Z 563.28,A -85,B 0,C 180,E1 9433.193,E2 9433.193} C_VEL
LIN {X 0,Y 417.733,Z 563.28,A -85,B 0,C 180,E1 9439.595,E2 9439.595} C_VEL
LIN {X 0,Y 418.005,Z 563.28,A -85,B 0,C 180,E1 9445.861,E2 9445.861} C_VEL
LIN {X 0,Y 418.201,Z 563.28,A -85,B 0,C 180,E1 9452.069,E2 9452.069} C_VEL
LIN {X 0,Y 417.783,Z 563.28,A -85,B 0,C 180,E1 9458.308,E2 9458.308} C_VEL
LIN {X 0,Y 417.55,Z 563.28,A -85,B 0,C 180,E1 9464.655,E2 9464.655} C_VEL
LIN {X 0,Y 417.335,Z 563.28,A -85,B 0,C 180,E1 9471.198,E2 9471.198} C_VEL
LIN {X 0,Y 417.015,Z 563.28,A -85,B 0,C 180,E1 9478.062,E2 9478.062} C_VEL
LIN {X 0,Y 416.972,Z 563.28,A -85,B 0,C 180,E1 9485.384,E2 9485.384} C_VEL
LIN {X 0,Y 416.945,Z 563.28,A -85,B 0,C 180,E1 9490.653,E2 9490.653} C_VEL
LIN {X 0,Y 416.919,Z 563.28,A -85,B 0,C 180,E1 9496.55,E2 9496.55} C_VEL
LIN {X 0,Y 417.002,Z 563.28,A -85,B 0,C 180,E1 9502.762,E2 9502.762} C_VEL
LIN {X 0,Y 417.031,Z 563.28,A -85,B 0,C 180,E1 9510.279,E2 9510.279} C_VEL
LIN {X 0,Y 417.236,Z 563.28,A -85,B 0,C 180,E1 9516.555,E2 9516.555} C_VEL
LIN {X 0,Y 417.425,Z 563.28,A -85,B 0,C 180,E1 9523.188,E2 9523.188} C_VEL
LIN {X 0,Y 417.587,Z 563.28,A -85,B 0,C 180,E1 9529.588,E2 9529.588} C_VEL
LIN {X 0,Y 417.947,Z 563.28,A -85,B 0,C 180,E1 9535.857,E2 9535.857} C_VEL
LIN {X 0,Y 417.981,Z 563.28,A -85,B 0,C 180,E1 9542.067,E2 9542.067} C_VEL
LIN {X 0,Y 417.774,Z 563.28,A -85,B 0,C 180,E1 9548.305,E2 9548.305} C_VEL
LIN {X 0,Y 417.593,Z 563.28,A -85,B 0,C 180,E1 9554.65,E2 9554.65} C_VEL
LIN {X 0,Y 417.339,Z 563.28,A -85,B 0,C 180,E1 9561.194,E2 9561.194} C_VEL
LIN {X 0,Y 417.082,Z 563.28,A -85,B 0,C 180,E1 9568.054,E2 9568.054} C_VEL
LIN {X 0,Y 417.047,Z 563.28,A -85,B 0,C 180,E1 9575.372,E2 9575.372} C_VEL
LIN {X 0,Y 416.901,Z 563.28,A -85,B 0,C 180,E1 9580.653,E2 9580.653} C_VEL
LIN {X 0,Y 416.819,Z 563.316,A -85,B 0,C 180,E1 9584.375,E2 9584.375} C_VEL
LIN {X 0,Y 419.192,Z 568.89,A -85,B 0,C 180,E1 9584.835,E2 9584.835} C_VEL
LIN {X 0,Y 441.265,Z 607.894,A -85,B 0,C 180,E1 9588.525,E2 9588.525} C_VEL
LIN {X 0,Y 449.745,Z 628.479,A -85,B 0,C 180,E1 9590.167,E2 9590.167} C_VEL
LIN {X 0,Y 445.571,Z 669.208,A -85,B 0,C 180,E1 9591.875,E2 9591.875} C_VEL
LIN {X 0,Y 440.459,Z 705.704,A -85,B 0,C 180,E1 9594.223,E2 9594.223} C_VEL
LIN {X 0,Y 434.69,Z 741.382,A -85,B 0,C 180,E1 9597.446,E2 9597.446} C_VEL
LIN {X 0,Y 428.756,Z 774.845,A -85,B 0,C 180,E1 9601.621,E2 9601.621} C_VEL
LIN {X 0,Y 424.272,Z 801.501,A -85,B 0,C 180,E1 9606.134,E2 9606.134} C_VEL
LIN {X 0,Y 422.485,Z 812.673,A -85,B 0,C 180,E1 9608.472,E2 9608.472} C_VEL
LIN {X 0,Y 417.451,Z 821.514,A -85,B 0,C 180,E1 9610.422,E2 9610.422} C_VEL
LIN {X 0,Y 412.468,Z 829.291,A -85,B 0,C 180,E1 9612.493,E2 9612.493} C_VEL
LIN {X 0,Y 411.024,Z 843.71,A -85,B 0,C 180,E1 9617.812,E2 9617.812} C_VEL
LIN {X 0,Y 410.485,Z 852.646,A -85,B 0,C 180,E1 9622.983,E2 9622.983} C_VEL
LIN {X 0,Y 410.336,Z 856.656,A -85,B 0,C 180,E1 9627.891,E2 9627.891} C_VEL
LIN {X 0,Y 410.366,Z 856.657,A -85,B 0,C 180,E1 9632.106,E2 9632.106} C_VEL
LIN {X 0,Y 410.528,Z 851.891,A -85,B 0,C 180,E1 9637.565,E2 9637.565} C_VEL
LIN {X 0,Y 411.119,Z 842.545,A -85,B 0,C 180,E1 9642.721,E2 9642.721} C_VEL
LIN {X 0,Y 412.629,Z 829.017,A -85,B 0,C 180,E1 9647.587,E2 9647.587} C_VEL
LIN {X 0,Y 415.948,Z 806.753,A -85,B 0,C 180,E1 9653.203,E2 9653.203} C_VEL
LIN {X 0,Y 420.298,Z 781.561,A -85,B 0,C 180,E1 9657.822,E2 9657.822} C_VEL
LIN {X 0,Y 425.814,Z 752.334,A -85,B 0,C 180,E1 9661.87,E2 9661.87} C_VEL
LIN {X 0,Y 431.917,Z 718.135,A -85,B 0,C 180,E1 9665.355,E2 9665.355} C_VEL
LIN {X 0,Y 437.488,Z 681.851,A -85,B 0,C 180,E1 9668.033,E2 9668.033} C_VEL
LIN {X 0,Y 442.431,Z 641.472,A -85,B 0,C 180,E1 9670.036,E2 9670.036} C_VEL
LIN {X 0,Y 443.002,Z 628.841,A -85,B 0,C 180,E1 9670.536,E2 9670.536} C_VEL
LIN {X 0,Y 427.206,Z 595.529,A -85,B 0,C 180,E1 9673.492,E2 9673.492} C_VEL
LIN {X 0,Y 409.019,Z 564.124,A -85,B 0,C 180,E1 9676.724,E2 9676.724} C_VEL
LIN {X 0,Y 408.886,Z 563.28,A -85,B 0,C 180,E1 9677.569,E2 9677.569} C_VEL
LIN {X 0,Y 409.007,Z 563.28,A -85,B 0,C 180,E1 9684.259,E2 9684.259} C_VEL
LIN {X 0,Y 409.086,Z 563.28,A -85,B 0,C 180,E1 9691.348,E2 9691.348} C_VEL
LIN {X 0,Y 409.366,Z 563.28,A -85,B 0,C 180,E1 9698.372,E2 9698.372} C_VEL
LIN {X 0,Y 409.471,Z 563.28,A -85,B 0,C 180,E1 9705.053,E2 9705.053} C_VEL
LIN {X 0,Y 409.807,Z 563.28,A -85,B 0,C 180,E1 9711.532,E2 9711.532} C_VEL
LIN {X 0,Y 410.268,Z 563.28,A -85,B 0,C 180,E1 9717.894,E2 9717.894} C_VEL
LIN {X 0,Y 410.075,Z 563.28,A -85,B 0,C 180,E1 9724.223,E2 9724.223} C_VEL
LIN {X 0,Y 409.782,Z 563.28,A -85,B 0,C 180,E1 9730.612,E2 9730.612} C_VEL
LIN {X 0,Y 409.563,Z 563.28,A -85,B 0,C 180,E1 9737.145,E2 9737.145} C_VEL
LIN {X 0,Y 409.301,Z 563.28,A -85,B 0,C 180,E1 9743.927,E2 9743.927} C_VEL
LIN {X 0,Y 409.117,Z 563.28,A -85,B 0,C 180,E1 9751.092,E2 9751.092} C_VEL
LIN {X 0,Y 409.106,Z 563.28,A -85,B 0,C 180,E1 9756.171,E2 9756.171} C_VEL
LIN {X 0,Y 408.847,Z 563.28,A -85,B 0,C 180,E1 9762.425,E2 9762.425} C_VEL
LIN {X 0,Y 408.868,Z 563.28,A -85,B 0,C 180,E1 9768.371,E2 9768.371} C_VEL
LIN {X 0,Y 409.143,Z 563.28,A -85,B 0,C 180,E1 9774.236,E2 9774.236} C_VEL
LIN {X 0,Y 409.183,Z 563.28,A -85,B 0,C 180,E1 9781.354,E2 9781.354} C_VEL
LIN {X 0,Y 409.318,Z 563.28,A -85,B 0,C 180,E1 9788.368,E2 9788.368} C_VEL
LIN {X 0,Y 409.644,Z 563.28,A -85,B 0,C 180,E1 9795.058,E2 9795.058} C_VEL
LIN {X 0,Y 409.865,Z 563.28,A -85,B 0,C 180,E1 9801.532,E2 9801.532} C_VEL
LIN {X 0,Y 410.141,Z 563.28,A -85,B 0,C 180,E1 9807.892,E2 9807.892} C_VEL
LIN {X 0,Y 410.052,Z 563.28,A -85,B 0,C 180,E1 9814.222,E2 9814.222} C_VEL
LIN {X 0,Y 409.769,Z 563.28,A -85,B 0,C 180,E1 9820.611,E2 9820.611} C_VEL
LIN {X 0,Y 409.538,Z 563.28,A -85,B 0,C 180,E1 9827.145,E2 9827.145} C_VEL
LIN {X 0,Y 409.273,Z 563.28,A -85,B 0,C 180,E1 9833.928,E2 9833.928} C_VEL
LIN {X 0,Y 408.994,Z 563.28,A -85,B 0,C 180,E1 9841.102,E2 9841.102} C_VEL
LIN {X 0,Y 409.061,Z 563.28,A -85,B 0,C 180,E1 9846.175,E2 9846.175} C_VEL
LIN {X 0,Y 408.923,Z 563.28,A -85,B 0,C 180,E1 9852.433,E2 9852.433} C_VEL
LIN {X 0,Y 408.916,Z 563.28,A -85,B 0,C 180,E1 9858.373,E2 9858.373} C_VEL
LIN {X 0,Y 409.017,Z 563.28,A -85,B 0,C 180,E1 9864.26,E2 9864.26} C_VEL
LIN {X 0,Y 409.089,Z 563.28,A -85,B 0,C 180,E1 9871.343,E2 9871.343} C_VEL
LIN {X 0,Y 409.384,Z 563.28,A -85,B 0,C 180,E1 9878.368,E2 9878.368} C_VEL
LIN {X 0,Y 409.475,Z 563.28,A -85,B 0,C 180,E1 9885.049,E2 9885.049} C_VEL
LIN {X 0,Y 409.821,Z 563.28,A -85,B 0,C 180,E1 9891.528,E2 9891.528} C_VEL
LIN {X 0,Y 410.285,Z 563.28,A -85,B 0,C 180,E1 9897.89,E2 9897.89} C_VEL
LIN {X 0,Y 410.061,Z 563.28,A -85,B 0,C 180,E1 9904.218,E2 9904.218} C_VEL
LIN {X 0,Y 409.806,Z 563.28,A -85,B 0,C 180,E1 9910.607,E2 9910.607} C_VEL
LIN {X 0,Y 409.554,Z 563.28,A -85,B 0,C 180,E1 9917.141,E2 9917.141} C_VEL
LIN {X 0,Y 409.287,Z 563.28,A -85,B 0,C 180,E1 9923.923,E2 9923.923} C_VEL
LIN {X 0,Y 409.113,Z 563.28,A -85,B 0,C 180,E1 9931.087,E2 9931.087} C_VEL
LIN {X 0,Y 409.097,Z 563.28,A -85,B 0,C 180,E1 9936.166,E2 9936.166} C_VEL
LIN {X 0,Y 408.893,Z 563.28,A -85,B 0,C 180,E1 9943.213,E2 9943.213} C_VEL
LIN {X 0,Y 411.469,Z 569.087,A -85,B 0,C 180,E1 9943.756,E2 9943.756} C_VEL
LIN {X 0,Y 433.916,Z 608.242,A -85,B 0,C 180,E1 9947.679,E2 9947.679} C_VEL
LIN {X 0,Y 443.483,Z 630.32,A -85,B 0,C 180,E1 9949.582,E2 9949.582} C_VEL
LIN {X 0,Y 439.231,Z 669.621,A -85,B 0,C 180,E1 9951.265,E2 9951.265} C_VEL
LIN {X 0,Y 433.673,Z 707.137,A -85,B 0,C 180,E1 9953.733,E2 9953.733} C_VEL
LIN {X 0,Y 427.636,Z 742.293,A -85,B 0,C 180,E1 9956.991,E2 9956.991} C_VEL
LIN {X 0,Y 421.609,Z 774.592,A -85,B 0,C 180,E1 9961.095,E2 9961.095} C_VEL
LIN {X 0,Y 416.725,Z 801.646,A -85,B 0,C 180,E1 9965.758,E2 9965.758} C_VEL
LIN {X 0,Y 413.321,Z 823.459,A -85,B 0,C 180,E1 9970.816,E2 9970.816} C_VEL
LIN {X 0,Y 412.468,Z 829.291,A -85,B 0,C 180,E1 9972.493,E2 9972.493} C_VEL
LIN {X 0,Y 407.768,Z 836.176,A -85,B 0,C 180,E1 9974.653,E2 9974.653} C_VEL
LIN {X 0,Y 403.276,Z 842.045,A -85,B 0,C 180,E1 9976.911,E2 9976.911} C_VEL
LIN {X 0,Y 402.693,Z 850.417,A -85,B 0,C 180,E1 9981.378,E2 9981.378} C_VEL
LIN {X 0,Y 402.446,Z 855.211,A -85,B 0,C 180,E1 9985.698,E2 9985.698} C_VEL
LIN {X 0,Y 402.457,Z 856.814,A -85,B 0,C 180,E1 9989.999,E2 9989.999} C_VEL
LIN {X 0,Y 402.438,Z 855.212,A -85,B 0,C 180,E1 9994.3,E2 9994.3} C_VEL
LIN {X 0,Y 402.755,Z 848.683,A -85,B 0,C 180,E1 9999.706,E2 9999.706} C_VEL
LIN {X 0,Y 403.823,Z 836.904,A -85,B 0,C 180,E1 10005.163,E2 10005.163} C_VEL
LIN {X 0,Y 406.12,Z 820.13,A -85,B 0,C 180,E1 10010.385,E2 10010.385} C_VEL
LIN {X 0,Y 410.233,Z 796.161,A -85,B 0,C 180,E1 10015.766,E2 10015.766} C_VEL
LIN {X 0,Y 415.955,Z 766.9,A -85,B 0,C 180,E1 10020.523,E2 10020.523} C_VEL
LIN {X 0,Y 422.017,Z 735.781,A -85,B 0,C 180,E1 10024.274,E2 10024.274} C_VEL
LIN {X 0,Y 428.411,Z 700.313,A -85,B 0,C 180,E1 10027.418,E2 10027.418} C_VEL
LIN {X 0,Y 433.851,Z 663.062,A -85,B 0,C 180,E1 10029.716,E2 10029.716} C_VEL
LIN {X 0,Y 436.689,Z 631.673,A -85,B 0,C 180,E1 10031.108,E2 10031.108} C_VEL
LIN {X 0,Y 421.437,Z 599.099,A -85,B 0,C 180,E1 10034.13,E2 10034.13} C_VEL
LIN {X 0,Y 402.987,Z 568.511,A -85,B 0,C 180,E1 10037.523,E2 10037.523} C_VEL
LIN {X 0,Y 400.978,Z 563.28,A -85,B 0,C 180,E1 10038.14,E2 10038.14} C_VEL
LIN {X 0,Y 400.987,Z 563.28,A -85,B 0,C 180,E1 10042.982,E2 10042.982} C_VEL
LIN {X 0,Y 401.054,Z 563.28,A -85,B 0,C 180,E1 10049.926,E2 10049.926} C_VEL
LIN {X 0,Y 401.284,Z 563.28,A -85,B 0,C 180,E1 10055.569,E2 10055.569} C_VEL
LIN {X 0,Y 401.551,Z 563.28,A -85,B 0,C 180,E1 10062.507,E2 10062.507} C_VEL
LIN {X 0,Y 401.738,Z 563.28,A -85,B 0,C 180,E1 10069.177,E2 10069.177} C_VEL
LIN {X 0,Y 402.129,Z 563.28,A -85,B 0,C 180,E1 10075.698,E2 10075.698} C_VEL
LIN {X 0,Y 402.251,Z 563.28,A -85,B 0,C 180,E1 10082.152,E2 10082.152} C_VEL
LIN {X 0,Y 401.91,Z 563.28,A -85,B 0,C 180,E1 10088.64,E2 10088.64} C_VEL
LIN {X 0,Y 401.73,Z 563.28,A -85,B 0,C 180,E1 10095.247,E2 10095.247} C_VEL
LIN {X 0,Y 401.445,Z 563.28,A -85,B 0,C 180,E1 10102.082,E2 10102.082} C_VEL
LIN {X 0,Y 401.2,Z 563.28,A -85,B 0,C 180,E1 10109.274,E2 10109.274} C_VEL
LIN {X 0,Y 401.189,Z 563.28,A -85,B 0,C 180,E1 10114.349,E2 10114.349} C_VEL
LIN {X 0,Y 400.943,Z 563.28,A -85,B 0,C 180,E1 10121.174,E2 10121.174} C_VEL
LIN {X 0,Y 400.928,Z 563.28,A -85,B 0,C 180,E1 10127.354,E2 10127.354} C_VEL
LIN {X 0,Y 401.077,Z 563.28,A -85,B 0,C 180,E1 10132.989,E2 10132.989} C_VEL
LIN {X 0,Y 401.176,Z 563.28,A -85,B 0,C 180,E1 10139.901,E2 10139.901} C_VEL
LIN {X 0,Y 401.277,Z 563.28,A -85,B 0,C 180,E1 10145.566,E2 10145.566} C_VEL
LIN {X 0,Y 401.584,Z 563.28,A -85,B 0,C 180,E1 10152.507,E2 10152.507} C_VEL
LIN {X 0,Y 401.89,Z 563.28,A -85,B 0,C 180,E1 10159.18,E2 10159.18} C_VEL
LIN {X 0,Y 402.191,Z 563.28,A -85,B 0,C 180,E1 10165.698,E2 10165.698} C_VEL
LIN {X 0,Y 402.402,Z 563.28,A -85,B 0,C 180,E1 10172.15,E2 10172.15} C_VEL
LIN {X 0,Y 401.926,Z 563.28,A -85,B 0,C 180,E1 10178.638,E2 10178.638} C_VEL
LIN {X 0,Y 401.693,Z 563.28,A -85,B 0,C 180,E1 10185.247,E2 10185.247} C_VEL
LIN {X 0,Y 401.418,Z 563.28,A -85,B 0,C 180,E1 10192.082,E2 10192.082} C_VEL
LIN {X 0,Y 401.083,Z 563.28,A -85,B 0,C 180,E1 10199.283,E2 10199.283} C_VEL
LIN {X 0,Y 401.097,Z 563.28,A -85,B 0,C 180,E1 10204.357,E2 10204.357} C_VEL
LIN {X 0,Y 400.989,Z 563.28,A -85,B 0,C 180,E1 10211.178,E2 10211.178} C_VEL
LIN {X 0,Y 401.002,Z 563.28,A -85,B 0,C 180,E1 10217.36,E2 10217.36} C_VEL
LIN {X 0,Y 401.009,Z 563.28,A -85,B 0,C 180,E1 10222.979,E2 10222.979} C_VEL
LIN {X 0,Y 401.064,Z 563.28,A -85,B 0,C 180,E1 10229.928,E2 10229.928} C_VEL
LIN {X 0,Y 401.304,Z 563.28,A -85,B 0,C 180,E1 10235.565,E2 10235.565} C_VEL
LIN {X 0,Y 401.568,Z 563.28,A -85,B 0,C 180,E1 10242.503,E2 10242.503} C_VEL
LIN {X 0,Y 401.74,Z 563.28,A -85,B 0,C 180,E1 10249.173,E2 10249.173} C_VEL
LIN {X 0,Y 402.143,Z 563.28,A -85,B 0,C 180,E1 10255.694,E2 10255.694} C_VEL
LIN {X 0,Y 402.332,Z 563.28,A -85,B 0,C 180,E1 10259.998,E2 10259.998} C_VEL
LIN {X 0,Y 402.073,Z 563.28,A -85,B 0,C 180,E1 10266.462,E2 10266.462} C_VEL
LIN {X 0,Y 401.844,Z 563.28,A -85,B 0,C 180,E1 10273.019,E2 10273.019} C_VEL
LIN {X 0,Y 401.469,Z 563.28,A -85,B 0,C 180,E1 10279.999,E2 10279.999} C_VEL
LIN {X 0,Y 401.257,Z 563.28,A -85,B 0,C 180,E1 10286.823,E2 10286.823} C_VEL
LIN {X 0,Y 401.179,Z 563.28,A -85,B 0,C 180,E1 10294.344,E2 10294.344} C_VEL
LIN {X 0,Y 400.927,Z 563.28,A -85,B 0,C 180,E1 10301.168,E2 10301.168} C_VEL
LIN {X 0,Y 400.987,Z 564,A -85,B 0,C 180,E1 10302.049,E2 10302.049} C_VEL
LIN {X 0,Y 403.624,Z 569.217,A -85,B 0,C 180,E1 10302.593,E2 10302.593} C_VEL
LIN {X 0,Y 425.498,Z 606.739,A -85,B 0,C 180,E1 10306.606,E2 10306.606} C_VEL
LIN {X 0,Y 437.199,Z 633.206,A -85,B 0,C 180,E1 10309.019,E2 10309.019} C_VEL
LIN {X 0,Y 432.79,Z 671.201,A -85,B 0,C 180,E1 10310.699,E2 10310.699} C_VEL
LIN {X 0,Y 426.661,Z 710.173,A -85,B 0,C 180,E1 10313.356,E2 10313.356} C_VEL
LIN {X 0,Y 420.358,Z 744.368,A -85,B 0,C 180,E1 10316.653,E2 10316.653} C_VEL
LIN {X 0,Y 414.132,Z 776.128,A -85,B 0,C 180,E1 10320.814,E2 10320.814} C_VEL
LIN {X 0,Y 408.824,Z 803.945,A -85,B 0,C 180,E1 10325.805,E2 10325.805} C_VEL
LIN {X 0,Y 405.323,Z 825.11,A -85,B 0,C 180,E1 10330.994,E2 10330.994} C_VEL
LIN {X 0,Y 403.367,Z 841.285,A -85,B 0,C 180,E1 10336.56,E2 10336.56} C_VEL
LIN {X 0,Y 403.276,Z 842.045,A -85,B 0,C 180,E1 10336.911,E2 10336.911} C_VEL
LIN {X 0,Y 398.951,Z 846.901,A -85,B 0,C 180,E1 10339.238,E2 10339.238} C_VEL
LIN {X 0,Y 394.753,Z 850.756,A -85,B 0,C 180,E1 10341.647,E2 10341.647} C_VEL
LIN {X 0,Y 394.541,Z 854.964,A -85,B 0,C 180,E1 10345.612,E2 10345.612} C_VEL
LIN {X 0,Y 394.56,Z 856.569,A -85,B 0,C 180,E1 10349.999,E2 10349.999} C_VEL
LIN {X 0,Y 394.534,Z 854.965,A -85,B 0,C 180,E1 10354.386,E2 10354.386} C_VEL
LIN {X 0,Y 394.885,Z 848.435,A -85,B 0,C 180,E1 10359.901,E2 10359.901} C_VEL
LIN {X 0,Y 396.028,Z 836.653,A -85,B 0,C 180,E1 10365.468,E2 10365.468} C_VEL
LIN {X 0,Y 398.469,Z 819.876,A -85,B 0,C 180,E1 10370.794,E2 10370.794} C_VEL
LIN {X 0,Y 402.795,Z 796.346,A -85,B 0,C 180,E1 10376.187,E2 10376.187} C_VEL
LIN {X 0,Y 408.901,Z 766.645,A -85,B 0,C 180,E1 10381.107,E2 10381.107} C_VEL
LIN {X 0,Y 415.484,Z 734.836,A -85,B 0,C 180,E1 10384.975,E2 10384.975} C_VEL
LIN {X 0,Y 422.183,Z 699.07,A -85,B 0,C 180,E1 10388.159,E2 10388.159} C_VEL
LIN {X 0,Y 427.996,Z 660.992,A -85,B 0,C 180,E1 10390.492,E2 10390.492} C_VEL
LIN {X 0,Y 430.496,Z 634.606,A -85,B 0,C 180,E1 10391.683,E2 10391.683} C_VEL
LIN {X 0,Y 415.19,Z 601.422,A -85,B 0,C 180,E1 10394.895,E2 10394.895} C_VEL
LIN {X 0,Y 395.584,Z 569.052,A -85,B 0,C 180,E1 10398.684,E2 10398.684} C_VEL
LIN {X 0,Y 393.203,Z 564.888,A -85,B 0,C 180,E1 10399.19,E2 10399.19} C_VEL
LIN {X 0,Y 393.04,Z 563.28,A -85,B 0,C 180,E1 10399.381,E2 10399.381} C_VEL
LIN {X 0,Y 393.024,Z 563.28,A -85,B 0,C 180,E1 10404.839,E2 10404.839} C_VEL
LIN {X 0,Y 393.17,Z 563.28,A -85,B 0,C 180,E1 10411.974,E2 10411.974} C_VEL
LIN {X 0,Y 393.437,Z 563.28,A -85,B 0,C 180,E1 10417.449,E2 10417.449} C_VEL
LIN {X 0,Y 393.638,Z 563.28,A -85,B 0,C 180,E1 10424.437,E2 10424.437} C_VEL
LIN {X 0,Y 393.953,Z 563.28,A -85,B 0,C 180,E1 10431.189,E2 10431.189} C_VEL
LIN {X 0,Y 394.468,Z 563.28,A -85,B 0,C 180,E1 10437.81,E2 10437.81} C_VEL
LIN {X 0,Y 394.26,Z 563.28,A -85,B 0,C 180,E1 10444.392,E2 10444.392} C_VEL
LIN {X 0,Y 393.929,Z 563.28,A -85,B 0,C 180,E1 10451.044,E2 10451.044} C_VEL
LIN {X 0,Y 393.659,Z 563.28,A -85,B 0,C 180,E1 10457.86,E2 10457.86} C_VEL
LIN {X 0,Y 393.388,Z 563.28,A -85,B 0,C 180,E1 10464.96,E2 10464.96} C_VEL
LIN {X 0,Y 393.241,Z 563.28,A -85,B 0,C 180,E1 10472.497,E2 10472.497} C_VEL
LIN {X 0,Y 393.117,Z 563.28,A -85,B 0,C 180,E1 10479.852,E2 10479.852} C_VEL
LIN {X 0,Y 393.013,Z 563.28,A -85,B 0,C 180,E1 10486.849,E2 10486.849} C_VEL
LIN {X 0,Y 393.144,Z 563.28,A -85,B 0,C 180,E1 10493.714,E2 10493.714} C_VEL
LIN {X 0,Y 393.305,Z 563.28,A -85,B 0,C 180,E1 10500.082,E2 10500.082} C_VEL
LIN {X 0,Y 393.411,Z 563.28,A -85,B 0,C 180,E1 10507.446,E2 10507.446} C_VEL
LIN {X 0,Y 393.768,Z 563.28,A -85,B 0,C 180,E1 10514.441,E2 10514.441} C_VEL
LIN {X 0,Y 394.023,Z 563.28,A -85,B 0,C 180,E1 10521.189,E2 10521.189} C_VEL
LIN {X 0,Y 394.34,Z 563.28,A -85,B 0,C 180,E1 10527.808,E2 10527.808} C_VEL
LIN {X 0,Y 394.249,Z 563.28,A -85,B 0,C 180,E1 10534.391,E2 10534.391} C_VEL
LIN {X 0,Y 393.917,Z 563.28,A -85,B 0,C 180,E1 10541.044,E2 10541.044} C_VEL
LIN {X 0,Y 393.635,Z 563.28,A -85,B 0,C 180,E1 10547.86,E2 10547.86} C_VEL
LIN {X 0,Y 393.345,Z 563.28,A -85,B 0,C 180,E1 10554.962,E2 10554.962} C_VEL
LIN {X 0,Y 393.152,Z 563.28,A -85,B 0,C 180,E1 10562.505,E2 10562.505} C_VEL
LIN {X 0,Y 393.134,Z 563.28,A -85,B 0,C 180,E1 10569.851,E2 10569.851} C_VEL
LIN {X 0,Y 393.084,Z 563.28,A -85,B 0,C 180,E1 10576.837,E2 10576.837} C_VEL
LIN {X 0,Y 393.054,Z 563.28,A -85,B 0,C 180,E1 10583.731,E2 10583.731} C_VEL
LIN {X 0,Y 393.164,Z 563.28,A -85,B 0,C 180,E1 10590.067,E2 10590.067} C_VEL
LIN {X 0,Y 393.46,Z 563.28,A -85,B 0,C 180,E1 10597.446,E2 10597.446} C_VEL
LIN {X 0,Y 393.648,Z 563.28,A -85,B 0,C 180,E1 10604.432,E2 10604.432} C_VEL
LIN {X 0,Y 393.965,Z 563.28,A -85,B 0,C 180,E1 10611.185,E2 10611.185} C_VEL
LIN {X 0,Y 394.483,Z 563.28,A -85,B 0,C 180,E1 10617.805,E2 10617.805} C_VEL
LIN {X 0,Y 394.25,Z 563.28,A -85,B 0,C 180,E1 10624.388,E2 10624.388} C_VEL
LIN {X 0,Y 393.953,Z 563.28,A -85,B 0,C 180,E1 10631.039,E2 10631.039} C_VEL
LIN {X 0,Y 393.646,Z 563.28,A -85,B 0,C 180,E1 10637.856,E2 10637.856} C_VEL
LIN {X 0,Y 393.372,Z 563.28,A -85,B 0,C 180,E1 10644.956,E2 10644.956} C_VEL
LIN {X 0,Y 393.237,Z 563.28,A -85,B 0,C 180,E1 10652.492,E2 10652.492} C_VEL
LIN {X 0,Y 393.1,Z 563.28,A -85,B 0,C 180,E1 10659.846,E2 10659.846} C_VEL
LIN {X 0,Y 393.04,Z 563.352,A -85,B 0,C 180,E1 10660.741,E2 10660.741} C_VEL
LIN {X 0,Y 395.281,Z 568.806,A -85,B 0,C 180,E1 10661.26,E2 10661.26} C_VEL
LIN {X 0,Y 416.028,Z 603.125,A -85,B 0,C 180,E1 10665.268,E2 10665.268} C_VEL
LIN {X 0,Y 430.873,Z 635.339,A -85,B 0,C 180,E1 10668.395,E2 10668.395} C_VEL
LIN {X 0,Y 426.256,Z 673.233,A -85,B 0,C 180,E1 10670.152,E2 10670.152} C_VEL
LIN {X 0,Y 419.924,Z 711.56,A -85,B 0,C 180,E1 10672.83,E2 10672.83} C_VEL
LIN {X 0,Y 413.306,Z 745.5,A -85,B 0,C 180,E1 10676.195,E2 10676.195} C_VEL
LIN {X 0,Y 406.948,Z 776.259,A -85,B 0,C 180,E1 10680.317,E2 10680.317} C_VEL
LIN {X 0,Y 401.168,Z 804.808,A -85,B 0,C 180,E1 10685.557,E2 10685.557} C_VEL
LIN {X 0,Y 397.434,Z 826.259,A -85,B 0,C 180,E1 10691.031,E2 10691.031} C_VEL
LIN {X 0,Y 395.527,Z 841.035,A -85,B 0,C 180,E1 10696.288,E2 10696.288} C_VEL
LIN {X 0,Y 394.753,Z 850.756,A -85,B 0,C 180,E1 10701.647,E2 10701.647} C_VEL
LIN {X 0,Y 392.083,Z 853.001,A -85,B 0,C 180,E1 10703.485,E2 10703.485} C_VEL
LIN {X 0,Y 386.668,Z 855.138,A -85,B 0,C 180,E1 10706.273,E2 10706.273} C_VEL
LIN {X 0,Y 386.574,Z 855.295,A -85,B 0,C 180,E1 10706.597,E2 10706.597} C_VEL
LIN {X 0,Y 386.663,Z 856.324,A -85,B 0,C 180,E1 10709.999,E2 10709.999} C_VEL
LIN {X 0,Y 386.644,Z 854.72,A -85,B 0,C 180,E1 10714.476,E2 10714.476} C_VEL
LIN {X 0,Y 387.013,Z 848.187,A -85,B 0,C 180,E1 10720.104,E2 10720.104} C_VEL
LIN {X 0,Y 388.245,Z 836.402,A -85,B 0,C 180,E1 10725.787,E2 10725.787} C_VEL
LIN {X 0,Y 390.962,Z 819.029,A -85,B 0,C 180,E1 10731.377,E2 10731.377} C_VEL
LIN {X 0,Y 395.506,Z 796.09,A -85,B 0,C 180,E1 10736.708,E2 10736.708} C_VEL
LIN {X 0,Y 401.918,Z 766.391,A -85,B 0,C 180,E1 10741.71,E2 10741.71} C_VEL
LIN {X 0,Y 408.697,Z 735.384,A -85,B 0,C 180,E1 10745.544,E2 10745.544} C_VEL
LIN {X 0,Y 415.583,Z 700.406,A -85,B 0,C 180,E1 10748.724,E2 10748.724} C_VEL
LIN {X 0,Y 421.451,Z 664.2,A -85,B 0,C 180,E1 10751.02,E2 10751.02} C_VEL
LIN {X 0,Y 424.358,Z 637.581,A -85,B 0,C 180,E1 10752.271,E2 10752.271} C_VEL
LIN {X 0,Y 409.831,Z 605.584,A -85,B 0,C 180,E1 10755.516,E2 10755.516} C_VEL
LIN {X 0,Y 391.354,Z 574.797,A -85,B 0,C 180,E1 10759.23,E2 10759.23} C_VEL
LIN {X 0,Y 385.224,Z 564.247,A -85,B 0,C 180,E1 10760.592,E2 10760.592} C_VEL
LIN {X 0,Y 385.154,Z 563.28,A -85,B 0,C 180,E1 10760.704,E2 10760.704} C_VEL
LIN {X 0,Y 385.105,Z 563.28,A -85,B 0,C 180,E1 10766.734,E2 10766.734} C_VEL
LIN {X 0,Y 385.33,Z 563.28,A -85,B 0,C 180,E1 10774.25,E2 10774.25} C_VEL
LIN {X 0,Y 385.649,Z 563.28,A -85,B 0,C 180,E1 10779.898,E2 10779.898} C_VEL
LIN {X 0,Y 385.792,Z 563.28,A -85,B 0,C 180,E1 10786.429,E2 10786.429} C_VEL
LIN {X 0,Y 386.223,Z 563.28,A -85,B 0,C 180,E1 10793.271,E2 10793.271} C_VEL
LIN {X 0,Y 386.523,Z 563.28,A -85,B 0,C 180,E1 10800.002,E2 10800.002} C_VEL
LIN {X 0,Y 386.218,Z 563.28,A -85,B 0,C 180,E1 10806.734,E2 10806.734} C_VEL
LIN {X 0,Y 385.933,Z 563.28,A -85,B 0,C 180,E1 10813.57,E2 10813.57} C_VEL
LIN {X 0,Y 385.611,Z 563.28,A -85,B 0,C 180,E1 10820.624,E2 10820.624} C_VEL
LIN {X 0,Y 385.377,Z 563.28,A -85,B 0,C 180,E1 10828.029,E2 10828.029} C_VEL
LIN {X 0,Y 385.214,Z 563.28,A -85,B 0,C 180,E1 10834.652,E2 10834.652} C_VEL
LIN {X 0,Y 385.217,Z 563.28,A -85,B 0,C 180,E1 10838.814,E2 10838.814} C_VEL
LIN {X 0,Y 385.006,Z 563.28,A -85,B 0,C 180,E1 10845.132,E2 10845.132} C_VEL
LIN {X 0,Y 385.208,Z 563.28,A -85,B 0,C 180,E1 10851.583,E2 10851.583} C_VEL
LIN {X 0,Y 385.24,Z 563.28,A -85,B 0,C 180,E1 10856.745,E2 10856.745} C_VEL
LIN {X 0,Y 385.36,Z 563.28,A -85,B 0,C 180,E1 10861.973,E2 10861.973} C_VEL
LIN {X 0,Y 385.566,Z 563.28,A -85,B 0,C 180,E1 10869.377,E2 10869.377} C_VEL
LIN {X 0,Y 385.945,Z 563.28,A -85,B 0,C 180,E1 10876.433,E2 10876.433} C_VEL
LIN {X 0,Y 386.249,Z 563.28,A -85,B 0,C 180,E1 10883.27,E2 10883.27} C_VEL
LIN {X 0,Y 386.533,Z 563.28,A -85,B 0,C 180,E1 10890.001,E2 10890.001} C_VEL
LIN {X 0,Y 386.268,Z 563.28,A -85,B 0,C 180,E1 10896.732,E2 10896.732} C_VEL
LIN {X 0,Y 385.916,Z 563.28,A -85,B 0,C 180,E1 10903.57,E2 10903.57} C_VEL
LIN {X 0,Y 385.589,Z 563.28,A -85,B 0,C 180,E1 10910.624,E2 10910.624} C_VEL
LIN {X 0,Y 385.27,Z 563.28,A -85,B 0,C 180,E1 10918.036,E2 10918.036} C_VEL
LIN {X 0,Y 385.182,Z 563.28,A -85,B 0,C 180,E1 10925.992,E2 10925.992} C_VEL
LIN {X 0,Y 385.102,Z 563.28,A -85,B 0,C 180,E1 10931.881,E2 10931.881} C_VEL
LIN {X 0,Y 385.096,Z 563.28,A -85,B 0,C 180,E1 10938.227,E2 10938.227} C_VEL
LIN {X 0,Y 385.143,Z 563.28,A -85,B 0,C 180,E1 10944.003,E2 10944.003} C_VEL
LIN {X 0,Y 385.283,Z 563.28,A -85,B 0,C 180,E1 10951.964,E2 10951.964} C_VEL
LIN {X 0,Y 385.614,Z 563.28,A -85,B 0,C 180,E1 10959.376,E2 10959.376} C_VEL
LIN {X 0,Y 385.777,Z 563.28,A -85,B 0,C 180,E1 10966.424,E2 10966.424} C_VEL
LIN {X 0,Y 386.243,Z 563.28,A -85,B 0,C 180,E1 10973.267,E2 10973.267} C_VEL
LIN {X 0,Y 386.527,Z 563.28,A -85,B 0,C 180,E1 10979.998,E2 10979.998} C_VEL
LIN {X 0,Y 386.23,Z 563.28,A -85,B 0,C 180,E1 10986.729,E2 10986.729} C_VEL
LIN {X 0,Y 385.979,Z 563.28,A -85,B 0,C 180,E1 10993.564,E2 10993.564} C_VEL
LIN {X 0,Y 385.594,Z 563.28,A -85,B 0,C 180,E1 11000.62,E2 11000.62} C_VEL
LIN {X 0,Y 385.367,Z 563.28,A -85,B 0,C 180,E1 11008.024,E2 11008.024} C_VEL
LIN {X 0,Y 385.205,Z 563.28,A -85,B 0,C 180,E1 11014.646,E2 11014.646} C_VEL
LIN {X 0,Y 385.242,Z 564.075,A -85,B 0,C 180,E1 11019.407,E2 11019.407} C_VEL
LIN {X 0,Y 388.158,Z 569.469,A -85,B 0,C 180,E1 11020.075,E2 11020.075} C_VEL
LIN {X 0,Y 410.671,Z 607.084,A -85,B 0,C 180,E1 11024.647,E2 11024.647} C_VEL
LIN {X 0,Y 424.658,Z 638.063,A -85,B 0,C 180,E1 11027.788,E2 11027.788} C_VEL
LIN {X 0,Y 419.586,Z 676.38,A -85,B 0,C 180,E1 11029.656,E2 11029.656} C_VEL
LIN {X 0,Y 413.227,Z 712.945,A -85,B 0,C 180,E1 11032.288,E2 11032.288} C_VEL
LIN {X 0,Y 406.047,Z 747.696,A -85,B 0,C 180,E1 11035.845,E2 11035.845} C_VEL
LIN {X 0,Y 399.532,Z 777.416,A -85,B 0,C 180,E1 11039.971,E2 11039.971} C_VEL
LIN {X 0,Y 393.754,Z 804.555,A -85,B 0,C 180,E1 11045.066,E2 11045.066} C_VEL
LIN {X 0,Y 389.983,Z 824.582,A -85,B 0,C 180,E1 11050.209,E2 11050.209} C_VEL
LIN {X 0,Y 387.72,Z 840.587,A -85,B 0,C 180,E1 11055.92,E2 11055.92} C_VEL
LIN {X 0,Y 386.851,Z 850.715,A -85,B 0,C 180,E1 11061.634,E2 11061.634} C_VEL
LIN {X 0,Y 386.574,Z 855.295,A -85,B 0,C 180,E1 11066.597,E2 11066.597} C_VEL
LIN {X 0,Y 384.041,Z 856.017,A -85,B 0,C 180,E1 11068.511,E2 11068.511} C_VEL
LIN {X 0,Y 378.782,Z 855.841,A -85,B 0,C 180,E1 11071.399,E2 11071.399} C_VEL
LIN {X 0,Y 378.712,Z 855.772,A -85,B 0,C 180,E1 11071.733,E2 11071.733} C_VEL
LIN {X 0,Y 378.867,Z 852.48,A -85,B 0,C 180,E1 11076.862,E2 11076.862} C_VEL
LIN {X 0,Y 379.514,Z 844.35,A -85,B 0,C 180,E1 11082.4,E2 11082.4} C_VEL
LIN {X 0,Y 381.498,Z 829.81,A -85,B 0,C 180,E1 11088.447,E2 11088.447} C_VEL
LIN {X 0,Y 385.088,Z 810.436,A -85,B 0,C 180,E1 11093.987,E2 11093.987} C_VEL
LIN {X 0,Y 390.405,Z 786.137,A -85,B 0,C 180,E1 11099.098,E2 11099.098} C_VEL
LIN {X 0,Y 397.428,Z 756.016,A -85,B 0,C 180,E1 11103.722,E2 11103.722} C_VEL
LIN {X 0,Y 404.462,Z 724.41,A -85,B 0,C 180,E1 11107.319,E2 11107.319} C_VEL
LIN {X 0,Y 411.744,Z 686.617,A -85,B 0,C 180,E1 11110.406,E2 11110.406} C_VEL
LIN {X 0,Y 417.55,Z 647.951,A -85,B 0,C 180,E1 11112.524,E2 11112.524} C_VEL
LIN {X 0,Y 417.999,Z 639.769,A -85,B 0,C 180,E1 11112.948,E2 11112.948} C_VEL
LIN {X 0,Y 403.166,Z 607.1,A -85,B 0,C 180,E1 11116.432,E2 11116.432} C_VEL
LIN {X 0,Y 383.983,Z 575.284,A -85,B 0,C 180,E1 11120.498,E2 11120.498} C_VEL
LIN {X 0,Y 377.406,Z 564.953,A -85,B 0,C 180,E1 11122.026,E2 11122.026} C_VEL
LIN {X 0,Y 377.195,Z 563.28,A -85,B 0,C 180,E1 11122.228,E2 11122.228} C_VEL
LIN {X 0,Y 377.192,Z 563.28,A -85,B 0,C 180,E1 11128.666,E2 11128.666} C_VEL
LIN {X 0,Y 377.39,Z 563.28,A -85,B 0,C 180,E1 11133.909,E2 11133.909} C_VEL
LIN {X 0,Y 377.619,Z 563.28,A -85,B 0,C 180,E1 11138.924,E2 11138.924} C_VEL
LIN {X 0,Y 377.847,Z 563.28,A -85,B 0,C 180,E1 11146.138,E2 11146.138} C_VEL
LIN {X 0,Y 378.301,Z 563.28,A -85,B 0,C 180,E1 11153.13,E2 11153.13} C_VEL
LIN {X 0,Y 378.621,Z 563.28,A -85,B 0,C 180,E1 11160.002,E2 11160.002} C_VEL
LIN {X 0,Y 378.301,Z 563.28,A -85,B 0,C 180,E1 11166.875,E2 11166.875} C_VEL
LIN {X 0,Y 377.985,Z 563.28,A -85,B 0,C 180,E1 11173.861,E2 11173.861} C_VEL
LIN {X 0,Y 377.642,Z 563.28,A -85,B 0,C 180,E1 11181.08,E2 11181.08} C_VEL
LIN {X 0,Y 377.399,Z 563.28,A -85,B 0,C 180,E1 11188.675,E2 11188.675} C_VEL
LIN {X 0,Y 377.295,Z 563.28,A -85,B 0,C 180,E1 11194.054,E2 11194.054} C_VEL
LIN {X 0,Y 377.115,Z 563.28,A -85,B 0,C 180,E1 11200.513,E2 11200.513} C_VEL
LIN {X 0,Y 377.036,Z 563.28,A -85,B 0,C 180,E1 11207.127,E2 11207.127} C_VEL
LIN {X 0,Y 377.257,Z 563.28,A -85,B 0,C 180,E1 11213.132,E2 11213.132} C_VEL
LIN {X 0,Y 377.331,Z 563.28,A -85,B 0,C 180,E1 11218.676,E2 11218.676} C_VEL
LIN {X 0,Y 377.416,Z 563.28,A -85,B 0,C 180,E1 11223.909,E2 11223.909} C_VEL
LIN {X 0,Y 377.727,Z 563.28,A -85,B 0,C 180,E1 11231.363,E2 11231.363} C_VEL
LIN {X 0,Y 378.134,Z 563.28,A -85,B 0,C 180,E1 11238.491,E2 11238.491} C_VEL
LIN {X 0,Y 378.467,Z 563.28,A -85,B 0,C 180,E1 11245.427,E2 11245.427} C_VEL
LIN {X 0,Y 378.664,Z 563.28,A -85,B 0,C 180,E1 11252.285,E2 11252.285} C_VEL
LIN {X 0,Y 378.144,Z 563.28,A -85,B 0,C 180,E1 11259.186,E2 11259.186} C_VEL
LIN {X 0,Y 377.803,Z 563.28,A -85,B 0,C 180,E1 11266.539,E2 11266.539} C_VEL
LIN {X 0,Y 377.523,Z 563.28,A -85,B 0,C 180,E1 11273.561,E2 11273.561} C_VEL
LIN {X 0,Y 377.315,Z 563.28,A -85,B 0,C 180,E1 11278.681,E2 11278.681} C_VEL
LIN {X 0,Y 377.216,Z 563.28,A -85,B 0,C 180,E1 11284.061,E2 11284.061} C_VEL
LIN {X 0,Y 377.135,Z 563.28,A -85,B 0,C 180,E1 11290.512,E2 11290.512} C_VEL
LIN {X 0,Y 377.093,Z 563.28,A -85,B 0,C 180,E1 11297.132,E2 11297.132} C_VEL
LIN {X 0,Y 377.18,Z 563.28,A -85,B 0,C 180,E1 11303.146,E2 11303.146} C_VEL
LIN {X 0,Y 377.185,Z 563.28,A -85,B 0,C 180,E1 11308.659,E2 11308.659} C_VEL
LIN {X 0,Y 377.403,Z 563.28,A -85,B 0,C 180,E1 11313.905,E2 11313.905} C_VEL
LIN {X 0,Y 377.643,Z 563.28,A -85,B 0,C 180,E1 11318.92,E2 11318.92} C_VEL
LIN {X 0,Y 377.836,Z 563.28,A -85,B 0,C 180,E1 11326.133,E2 11326.133} C_VEL
LIN {X 0,Y 378.319,Z 563.28,A -85,B 0,C 180,E1 11333.13,E2 11333.13} C_VEL
LIN {X 0,Y 378.625,Z 563.28,A -85,B 0,C 180,E1 11339.998,E2 11339.998} C_VEL
LIN {X 0,Y 378.312,Z 563.28,A -85,B 0,C 180,E1 11346.87,E2 11346.87} C_VEL
LIN {X 0,Y 378.025,Z 563.28,A -85,B 0,C 180,E1 11353.855,E2 11353.855} C_VEL
LIN {X 0,Y 377.625,Z 563.28,A -85,B 0,C 180,E1 11361.075,E2 11361.075} C_VEL
LIN {X 0,Y 377.391,Z 563.28,A -85,B 0,C 180,E1 11368.671,E2 11368.671} C_VEL
LIN {X 0,Y 377.287,Z 563.28,A -85,B 0,C 180,E1 11374.049,E2 11374.049} C_VEL
LIN {X 0,Y 377.284,Z 563.861,A -85,B 0,C 180,E1 11377.917,E2 11377.917} C_VEL
LIN {X 0,Y 380.186,Z 569.384,A -85,B 0,C 180,E1 11378.634,E2 11378.634} C_VEL
LIN {X 0,Y 401.141,Z 603.657,A -85,B 0,C 180,E1 11383.158,E2 11383.158} C_VEL
LIN {X 0,Y 416.826,Z 636.589,A -85,B 0,C 180,E1 11386.747,E2 11386.747} C_VEL
LIN {X 0,Y 418.395,Z 642.214,A -85,B 0,C 180,E1 11387.241,E2 11387.241} C_VEL
LIN {X 0,Y 412.725,Z 681.487,A -85,B 0,C 180,E1 11389.276,E2 11389.276} C_VEL
LIN {X 0,Y 405.938,Z 717.107,A -85,B 0,C 180,E1 11391.997,E2 11391.997} C_VEL
LIN {X 0,Y 398.534,Z 751.166,A -85,B 0,C 180,E1 11395.636,E2 11395.636} C_VEL
LIN {X 0,Y 391.446,Z 781.447,A -85,B 0,C 180,E1 11400.096,E2 11400.096} C_VEL
LIN {X 0,Y 385.806,Z 806.797,A -85,B 0,C 180,E1 11405.135,E2 11405.135} C_VEL
LIN {X 0,Y 381.692,Z 828.093,A -85,B 0,C 180,E1 11410.963,E2 11410.963} C_VEL
LIN {X 0,Y 379.655,Z 842.506,A -85,B 0,C 180,E1 11416.685,E2 11416.685} C_VEL
LIN {X 0,Y 378.958,Z 851.14,A -85,B 0,C 180,E1 11421.988,E2 11421.988} C_VEL
LIN {X 0,Y 378.743,Z 855.674,A -85,B 0,C 180,E1 11427.716,E2 11427.716} C_VEL
LIN {X 0,Y 378.712,Z 855.772,A -85,B 0,C 180,E1 11431.733,E2 11431.733} C_VEL
LIN {X 0,Y 376.22,Z 854.953,A -85,B 0,C 180,E1 11433.682,E2 11433.682} C_VEL
LIN {X 0,Y 370.999,Z 852.592,A -85,B 0,C 180,E1 11436.606,E2 11436.606} C_VEL
LIN {X 0,Y 370.96,Z 852.288,A -85,B 0,C 180,E1 11436.944,E2 11436.944} C_VEL
LIN {X 0,Y 371.715,Z 843.378,A -85,B 0,C 180,E1 11443.032,E2 11443.032} C_VEL
LIN {X 0,Y 373.762,Z 829.556,A -85,B 0,C 180,E1 11448.843,E2 11448.843} C_VEL
LIN {X 0,Y 377.544,Z 810.179,A -85,B 0,C 180,E1 11454.498,E2 11454.498} C_VEL
LIN {X 0,Y 383.555,Z 784.55,A -85,B 0,C 180,E1 11459.936,E2 11459.936} C_VEL
LIN {X 0,Y 391.209,Z 753.609,A -85,B 0,C 180,E1 11464.678,E2 11464.678} C_VEL
LIN {X 0,Y 398.671,Z 721.322,A -85,B 0,C 180,E1 11468.292,E2 11468.292} C_VEL
LIN {X 0,Y 406.071,Z 684.457,A -85,B 0,C 180,E1 11471.269,E2 11471.269} C_VEL
LIN {X 0,Y 411.953,Z 643.031,A -85,B 0,C 180,E1 11473.526,E2 11473.526} C_VEL
LIN {X 0,Y 397.257,Z 610.186,A -85,B 0,C 180,E1 11477.205,E2 11477.205} C_VEL
LIN {X 0,Y 379.585,Z 580.612,A -85,B 0,C 180,E1 11481.147,E2 11481.147} C_VEL
LIN {X 0,Y 371.28,Z 568.541,A -85,B 0,C 180,E1 11483.131,E2 11483.131} C_VEL
LIN {X 0,Y 369.205,Z 563.28,A -85,B 0,C 180,E1 11483.919,E2 11483.919} C_VEL
LIN {X 0,Y 369.305,Z 563.28,A -85,B 0,C 180,E1 11490.641,E2 11490.641} C_VEL
LIN {X 0,Y 369.527,Z 563.28,A -85,B 0,C 180,E1 11495.901,E2 11495.901} C_VEL
LIN {X 0,Y 369.839,Z 563.28,A -85,B 0,C 180,E1 11503.407,E2 11503.407} C_VEL
LIN {X 0,Y 370.144,Z 563.28,A -85,B 0,C 180,E1 11510.617,E2 11510.617} C_VEL
LIN {X 0,Y 370.74,Z 563.28,A -85,B 0,C 180,E1 11517.67,E2 11517.67} C_VEL
LIN {X 0,Y 370.531,Z 563.28,A -85,B 0,C 180,E1 11524.674,E2 11524.674} C_VEL
LIN {X 0,Y 370.162,Z 563.28,A -85,B 0,C 180,E1 11531.938,E2 11531.938} C_VEL
LIN {X 0,Y 369.792,Z 563.28,A -85,B 0,C 180,E1 11539.056,E2 11539.056} C_VEL
LIN {X 0,Y 369.497,Z 563.28,A -85,B 0,C 180,E1 11546.697,E2 11546.697} C_VEL
LIN {X 0,Y 369.393,Z 563.28,A -85,B 0,C 180,E1 11552.08,E2 11552.08} C_VEL
LIN {X 0,Y 369.18,Z 563.28,A -85,B 0,C 180,E1 11559.05,E2 11559.05} C_VEL
LIN {X 0,Y 369.122,Z 563.28,A -85,B 0,C 180,E1 11565.976,E2 11565.976} C_VEL
LIN {X 0,Y 369.213,Z 563.28,A -85,B 0,C 180,E1 11572.19,E2 11572.19} C_VEL
LIN {X 0,Y 369.418,Z 563.28,A -85,B 0,C 180,E1 11579.075,E2 11579.075} C_VEL
LIN {X 0,Y 369.529,Z 563.28,A -85,B 0,C 180,E1 11585.899,E2 11585.899} C_VEL
LIN {X 0,Y 369.915,Z 563.28,A -85,B 0,C 180,E1 11593.409,E2 11593.409} C_VEL
LIN {X 0,Y 370.238,Z 563.28,A -85,B 0,C 180,E1 11600.618,E2 11600.618} C_VEL
LIN {X 0,Y 370.642,Z 563.28,A -85,B 0,C 180,E1 11607.668,E2 11607.668} C_VEL
LIN {X 0,Y 370.761,Z 563.28,A -85,B 0,C 180,E1 11612.334,E2 11612.334} C_VEL
LIN {X 0,Y 370.214,Z 563.28,A -85,B 0,C 180,E1 11619.385,E2 11619.385} C_VEL
LIN {X 0,Y 369.903,Z 563.28,A -85,B 0,C 180,E1 11626.594,E2 11626.594} C_VEL
LIN {X 0,Y 369.532,Z 563.28,A -85,B 0,C 180,E1 11634.103,E2 11634.103} C_VEL
LIN {X 0,Y 369.268,Z 563.28,A -85,B 0,C 180,E1 11642.091,E2 11642.091} C_VEL
LIN {X 0,Y 369.177,Z 563.28,A -85,B 0,C 180,E1 11649.045,E2 11649.045} C_VEL
LIN {X 0,Y 369.188,Z 563.28,A -85,B 0,C 180,E1 11655.982,E2 11655.982} C_VEL
LIN {X 0,Y 369.159,Z 563.28,A -85,B 0,C 180,E1 11662.18,E2 11662.18} C_VEL
LIN {X 0,Y 369.272,Z 563.28,A -85,B 0,C 180,E1 11669.112,E2 11669.112} C_VEL
LIN {X 0,Y 369.547,Z 563.28,A -85,B 0,C 180,E1 11675.897,E2 11675.897} C_VEL
LIN {X 0,Y 369.778,Z 563.28,A -85,B 0,C 180,E1 11680.943,E2 11680.943} C_VEL
LIN {X 0,Y 370.021,Z 563.28,A -85,B 0,C 180,E1 11688.232,E2 11688.232} C_VEL
LIN {X 0,Y 370.509,Z 563.28,A -85,B 0,C 180,E1 11695.325,E2 11695.325} C_VEL
LIN {X 0,Y 370.747,Z 563.28,A -85,B 0,C 180,E1 11699.998,E2 11699.998} C_VEL
LIN {X 0,Y 370.381,Z 563.28,A -85,B 0,C 180,E1 11707.018,E2 11707.018} C_VEL
LIN {X 0,Y 370.098,Z 563.28,A -85,B 0,C 180,E1 11714.158,E2 11714.158} C_VEL
LIN {X 0,Y 369.685,Z 563.28,A -85,B 0,C 180,E1 11721.55,E2 11721.55} C_VEL
LIN {X 0,Y 369.487,Z 563.28,A -85,B 0,C 180,E1 11726.692,E2 11726.692} C_VEL
LIN {X 0,Y 369.388,Z 563.28,A -85,B 0,C 180,E1 11732.074,E2 11732.074} C_VEL
LIN {X 0,Y 369.3,Z 563.28,A -85,B 0,C 180,E1 11736.265,E2 11736.265} C_VEL
LIN {X 0,Y 371.562,Z 568.767,A -85,B 0,C 180,E1 11736.933,E2 11736.933} C_VEL
LIN {X 0,Y 385.881,Z 590.601,A -85,B 0,C 180,E1 11740.272,E2 11740.272} C_VEL
LIN {X 0,Y 402.922,Z 621.538,A -85,B 0,C 180,E1 11744.123,E2 11744.123} C_VEL
LIN {X 0,Y 412.213,Z 643.595,A -85,B 0,C 180,E1 11746.541,E2 11746.541} C_VEL
LIN {X 0,Y 406.329,Z 683.371,A -85,B 0,C 180,E1 11748.672,E2 11748.672} C_VEL
LIN {X 0,Y 398.91,Z 719.939,A -85,B 0,C 180,E1 11751.571,E2 11751.571} C_VEL
LIN {X 0,Y 391.55,Z 752.15,A -85,B 0,C 180,E1 11755.122,E2 11755.122} C_VEL
LIN {X 0,Y 383.863,Z 783.347,A -85,B 0,C 180,E1 11759.859,E2 11759.859} C_VEL
LIN {X 0,Y 378.117,Z 807.752,A -85,B 0,C 180,E1 11764.91,E2 11764.91} C_VEL
LIN {X 0,Y 374.002,Z 827.84,A -85,B 0,C 180,E1 11770.556,E2 11770.556} C_VEL
LIN {X 0,Y 371.802,Z 842.541,A -85,B 0,C 180,E1 11776.544,E2 11776.544} C_VEL
LIN {X 0,Y 371.063,Z 850.892,A -85,B 0,C 180,E1 11781.816,E2 11781.816} C_VEL
LIN {X 0,Y 370.868,Z 855.43,A -85,B 0,C 180,E1 11787.667,E2 11787.667} C_VEL
LIN {X 0,Y 370.89,Z 855.431,A -85,B 0,C 180,E1 11792.331,E2 11792.331} C_VEL
LIN {X 0,Y 370.96,Z 852.288,A -85,B 0,C 180,E1 11796.944,E2 11796.944} C_VEL
LIN {X 0,Y 368.687,Z 850.141,A -85,B 0,C 180,E1 11798.915,E2 11798.915} C_VEL
LIN {X 0,Y 363.7,Z 845.741,A -85,B 0,C 180,E1 11801.853,E2 11801.853} C_VEL
LIN {X 0,Y 363.671,Z 845.185,A -85,B 0,C 180,E1 11802.19,E2 11802.19} C_VEL
LIN {X 0,Y 365.656,Z 831.716,A -85,B 0,C 180,E1 11808.356,E2 11808.356} C_VEL
LIN {X 0,Y 369.663,Z 812.346,A -85,B 0,C 180,E1 11814.412,E2 11814.412} C_VEL
LIN {X 0,Y 375.916,Z 786.459,A -85,B 0,C 180,E1 11820.152,E2 11820.152} C_VEL
LIN {X 0,Y 383.488,Z 757.412,A -85,B 0,C 180,E1 11824.811,E2 11824.811} C_VEL
LIN {X 0,Y 391.652,Z 724.346,A -85,B 0,C 180,E1 11828.709,E2 11828.709} C_VEL
LIN {X 0,Y 399.686,Z 686.11,A -85,B 0,C 180,E1 11831.895,E2 11831.895} C_VEL
LIN {X 0,Y 405.956,Z 647.506,A -85,B 0,C 180,E1 11834.04,E2 11834.04} C_VEL
LIN {X 0,Y 395.255,Z 620.886,A -85,B 0,C 180,E1 11837.048,E2 11837.048} C_VEL
LIN {X 0,Y 379.629,Z 592.56,A -85,B 0,C 180,E1 11840.786,E2 11840.786} C_VEL
LIN {X 0,Y 364.349,Z 569.547,A -85,B 0,C 180,E1 11844.565,E2 11844.565} C_VEL
LIN {X 0,Y 361.46,Z 565.022,A -85,B 0,C 180,E1 11845.362,E2 11845.362} C_VEL
LIN {X 0,Y 361.257,Z 563.28,A -85,B 0,C 180,E1 11845.499,E2 11845.499} C_VEL
LIN {X 0,Y 361.434,Z 563.28,A -85,B 0,C 180,E1 11852.664,E2 11852.664} C_VEL
LIN {X 0,Y 361.689,Z 563.28,A -85,B 0,C 180,E1 11857.948,E2 11857.948} C_VEL
LIN {X 0,Y 361.972,Z 563.28,A -85,B 0,C 180,E1 11865.518,E2 11865.518} C_VEL
LIN {X 0,Y 362.446,Z 563.28,A -85,B 0,C 180,E1 11872.828,E2 11872.828} C_VEL
LIN {X 0,Y 362.842,Z 563.28,A -85,B 0,C 180,E1 11880.003,E2 11880.003} C_VEL
LIN {X 0,Y 362.455,Z 563.28,A -85,B 0,C 180,E1 11887.177,E2 11887.177} C_VEL
LIN {X 0,Y 362.091,Z 563.28,A -85,B 0,C 180,E1 11894.483,E2 11894.483} C_VEL
LIN {X 0,Y 361.716,Z 563.28,A -85,B 0,C 180,E1 11902.055,E2 11902.055} C_VEL
LIN {X 0,Y 361.475,Z 563.28,A -85,B 0,C 180,E1 11910.065,E2 11910.065} C_VEL
LIN {X 0,Y 361.276,Z 563.28,A -85,B 0,C 180,E1 11917.478,E2 11917.478} C_VEL
LIN {X 0,Y 361.18,Z 563.28,A -85,B 0,C 180,E1 11924.746,E2 11924.746} C_VEL
LIN {X 0,Y 361.274,Z 563.28,A -85,B 0,C 180,E1 11931.206,E2 11931.206} C_VEL
LIN {X 0,Y 361.378,Z 563.28,A -85,B 0,C 180,E1 11937.124,E2 11937.124} C_VEL
LIN {X 0,Y 361.484,Z 563.28,A -85,B 0,C 180,E1 11942.666,E2 11942.666} C_VEL
LIN {X 0,Y 361.645,Z 564.04,A -85,B 0,C 180,E1 11945.698,E2 11945.698} C_VEL
LIN {X 0,Y 363.032,Z 567.591,A -85,B 0,C 180,E1 11949.112,E2 11949.112} C_VEL
LIN {X 0,Y 365.511,Z 569.768,A -85,B 0,C 180,E1 11955.659,E2 11955.659} C_VEL
LIN {X 0,Y 366.871,Z 570.431,A -85,B 0,C 180,E1 11960.82,E2 11960.82} C_VEL
LIN {X 0,Y 367.828,Z 570.662,A -85,B 0,C 180,E1 11967.65,E2 11967.65} C_VEL
LIN {X 0,Y 367.629,Z 570.634,A -85,B 0,C 180,E1 11974.71,E2 11974.71} C_VEL
LIN {X 0,Y 366.249,Z 570.138,A -85,B 0,C 180,E1 11981.89,E2 11981.89} C_VEL
LIN {X 0,Y 363.927,Z 568.621,A -85,B 0,C 180,E1 11988.746,E2 11988.746} C_VEL
LIN {X 0,Y 361.743,Z 564.532,A -85,B 0,C 180,E1 11994.029,E2 11994.029} C_VEL
LIN {X 0,Y 361.597,Z 563.28,A -85,B 0,C 180,E1 11994.667,E2 11994.667} C_VEL
LIN {X 0,Y 361.364,Z 563.28,A -85,B 0,C 180,E1 12000.074,E2 12000.074} C_VEL
LIN {X 0,Y 361.253,Z 563.28,A -85,B 0,C 180,E1 12007.468,E2 12007.468} C_VEL
LIN {X 0,Y 361.267,Z 563.28,A -85,B 0,C 180,E1 12014.755,E2 12014.755} C_VEL
LIN {X 0,Y 361.242,Z 563.28,A -85,B 0,C 180,E1 12021.198,E2 12021.198} C_VEL
LIN {X 0,Y 361.236,Z 563.28,A -85,B 0,C 180,E1 12027.106,E2 12027.106} C_VEL
LIN {X 0,Y 361.441,Z 563.28,A -85,B 0,C 180,E1 12032.659,E2 12032.659} C_VEL
LIN {X 0,Y 361.713,Z 563.28,A -85,B 0,C 180,E1 12037.945,E2 12037.945} C_VEL
LIN {X 0,Y 361.949,Z 563.28,A -85,B 0,C 180,E1 12045.511,E2 12045.511} C_VEL
LIN {X 0,Y 362.447,Z 563.28,A -85,B 0,C 180,E1 12053.11,E2 12053.11} C_VEL
LIN {X 0,Y 362.844,Z 563.28,A -85,B 0,C 180,E1 12059.997,E2 12059.997} C_VEL
LIN {X 0,Y 362.467,Z 563.28,A -85,B 0,C 180,E1 12067.172,E2 12067.172} C_VEL
LIN {X 0,Y 362.136,Z 563.28,A -85,B 0,C 180,E1 12074.476,E2 12074.476} C_VEL
LIN {X 0,Y 361.7,Z 563.28,A -85,B 0,C 180,E1 12082.051,E2 12082.051} C_VEL
LIN {X 0,Y 361.468,Z 563.28,A -85,B 0,C 180,E1 12090.06,E2 12090.06} C_VEL
LIN {X 0,Y 361.391,Z 563.911,A -85,B 0,C 180,E1 12094.584,E2 12094.584} C_VEL
LIN {X 0,Y 364.141,Z 569.259,A -85,B 0,C 180,E1 12095.38,E2 12095.38} C_VEL
LIN {X 0,Y 378.847,Z 591.453,A -85,B 0,C 180,E1 12099.034,E2 12099.034} C_VEL
LIN {X 0,Y 396.124,Z 622.598,A -85,B 0,C 180,E1 12103.159,E2 12103.159} C_VEL
LIN {X 0,Y 406.052,Z 646.406,A -85,B 0,C 180,E1 12105.904,E2 12105.904} C_VEL
LIN {X 0,Y 400.157,Z 684.18,A -85,B 0,C 180,E1 12107.981,E2 12107.981} C_VEL
LIN {X 0,Y 392.161,Z 721.759,A -85,B 0,C 180,E1 12111.037,E2 12111.037} C_VEL
LIN {X 0,Y 384.276,Z 754.236,A -85,B 0,C 180,E1 12114.749,E2 12114.749} C_VEL
LIN {X 0,Y 376.245,Z 785.387,A -85,B 0,C 180,E1 12119.642,E2 12119.642} C_VEL
LIN {X 0,Y 369.877,Z 811.126,A -85,B 0,C 180,E1 12125.279,E2 12125.279} C_VEL
LIN {X 0,Y 366.01,Z 829.295,A -85,B 0,C 180,E1 12130.74,E2 12130.74} C_VEL
LIN {X 0,Y 363.869,Z 843.133,A -85,B 0,C 180,E1 12136.685,E2 12136.685} C_VEL
LIN {X 0,Y 363.087,Z 851.984,A -85,B 0,C 180,E1 12142.837,E2 12142.837} C_VEL
LIN {X 0,Y 362.963,Z 855.184,A -85,B 0,C 180,E1 12147.616,E2 12147.616} C_VEL
LIN {X 0,Y 362.984,Z 855.185,A -85,B 0,C 180,E1 12152.381,E2 12152.381} C_VEL
LIN {X 0,Y 363.184,Z 850.648,A -85,B 0,C 180,E1 12158.361,E2 12158.361} C_VEL
